C09108=1129.768,245.322,-69.072,-178.598,9.848,149.571
C09109=1129.764,245.570,-69.100,-178.596,9.851,149.571
C09110=1129.759,245.818,-69.127,-178.595,9.853,149.572
C09111=1129.756,246.067,-69.155,-178.594,9.855,149.572
C09112=1129.751,246.315,-69.183,-178.593,9.857,149.572
C09113=1129.747,246.564,-69.212,-178.591,9.859,149.572
C09114=1129.742,246.812,-69.239,-178.590,9.861,149.572
C09115=1129.738,247.060,-69.266,-178.588,9.864,149.572
C09116=1129.734,247.309,-69.295,-178.587,9.865,149.572
C09117=1129.729,247.557,-69.322,-178.583,9.870,149.572
C09118=1129.725,247.806,-69.350,-178.576,9.875,149.572
C09119=1129.721,248.054,-69.378,-178.568,9.881,149.571
C09120=1129.716,248.302,-69.406,-178.562,9.886,149.571
C09121=1129.711,248.551,-69.434,-178.555,9.891,149.570
C09122=1129.707,248.799,-69.462,-178.549,9.896,149.570
C09123=1129.703,249.048,-69.490,-178.543,9.900,149.569
C09124=1129.698,249.296,-69.518,-178.537,9.905,149.568
C09125=1129.694,249.545,-69.546,-178.532,9.909,149.568
C09126=1129.690,249.792,-69.574,-178.526,9.913,149.568
C09127=1129.686,250.041,-69.603,-178.521,9.917,149.567
C09128=1129.682,250.290,-69.631,-178.516,9.921,149.567
C09129=1129.678,250.538,-69.659,-178.512,9.925,149.567
C09130=1129.673,250.787,-69.688,-178.507,9.928,149.566
C09131=1129.669,251.034,-69.715,-178.503,9.931,149.566
C09132=1129.664,251.283,-69.744,-178.499,9.934,149.565
C09133=1129.660,251.531,-69.772,-178.495,9.937,149.565
C09134=1129.656,251.780,-69.801,-178.492,9.940,149.565
C09135=1129.652,252.028,-69.829,-178.488,9.943,149.565
C09136=1129.648,252.276,-69.857,-178.486,9.945,149.565
C09137=1129.643,252.525,-69.886,-178.483,9.947,149.565
C09138=1129.639,252.739,-69.910,-178.481,9.949,149.564
C09139=1129.635,252.953,-69.935,-178.479,9.951,149.564
C09140=1129.633,253.166,-69.960,-178.477,9.953,149.564
C09141=1129.628,253.379,-69.984,-178.476,9.955,149.564
C09142=1129.624,253.593,-70.008,-178.474,9.956,149.564
C09143=1129.620,253.807,-70.033,-178.474,9.957,149.564
C09144=1129.617,254.021,-70.058,-178.472,9.958,149.564
C09145=1129.613,254.235,-70.082,-178.472,9.959,149.564
C09146=1129.609,254.484,-70.110,-178.471,9.961,149.565
C09147=1129.605,254.732,-70.139,-178.471,9.962,149.565
C09148=1129.600,254.980,-70.167,-178.470,9.963,149.565
C09149=1129.596,255.229,-70.196,-178.471,9.963,149.565
C09150=1129.592,255.476,-70.224,-178.471,9.965,149.566
C09151=1129.587,255.725,-70.253,-178.472,9.966,149.566
C09152=1129.583,255.974,-70.281,-178.472,9.966,149.566
C09153=1129.579,256.221,-70.310,-178.469,9.969,149.566
C09154=1129.575,256.470,-70.338,-178.467,9.972,149.566
C09155=1129.570,256.719,-70.367,-178.464,9.975,149.566
C09156=1129.566,256.967,-70.395,-178.461,9.977,149.566
C09157=1129.562,257.215,-70.424,-178.458,9.980,149.566
C09158=1129.557,257.464,-70.453,-178.455,9.983,149.566
C09159=1129.553,257.712,-70.481,-178.451,9.986,149.566
C09160=1129.549,257.960,-70.510,-178.448,9.989,149.565
C09161=1129.545,258.209,-70.538,-178.446,9.992,149.565
C09162=1129.540,258.457,-70.567,-178.443,9.995,149.565
C09163=1129.536,258.705,-70.596,-178.439,9.998,149.565
C09164=1129.532,258.954,-70.624,-178.436,10.001,149.565
C09165=1129.527,259.201,-70.653,-178.433,10.004,149.565
C09166=1129.523,259.450,-70.682,-178.430,10.007,149.565
C09167=1129.519,259.698,-70.711,-178.427,10.010,149.565
C09168=1129.514,259.946,-70.739,-178.423,10.013,149.564
C09169=1129.510,260.195,-70.769,-178.420,10.016,149.564
C09170=1129.506,260.443,-70.797,-178.416,10.019,149.564
C09171=1129.502,260.691,-70.826,-178.413,10.022,149.564
C09172=1129.497,260.940,-70.855,-178.409,10.025,149.564
C09173=1129.493,261.188,-70.884,-178.406,10.028,149.564
C09174=1129.489,261.436,-70.912,-178.402,10.031,149.563
C09175=1129.485,261.685,-70.942,-178.399,10.034,149.563
C09176=1129.480,261.933,-70.970,-178.395,10.037,149.563
C09177=1129.476,262.181,-71.000,-178.392,10.041,149.563
C09178=1129.472,262.429,-71.028,-178.388,10.044,149.563
C09179=1129.468,262.678,-71.057,-178.385,10.047,149.563
C09180=1129.463,262.926,-71.086,-178.381,10.050,149.562
C09181=1129.459,263.174,-71.115,-178.377,10.053,149.562
C09182=1129.454,263.423,-71.144,-178.373,10.056,149.562
C09183=1129.451,263.671,-71.173,-178.369,10.060,149.562
C09184=1129.447,263.919,-71.203,-178.366,10.062,149.561
C09185=1129.442,264.168,-71.232,-178.362,10.065,149.561
C09186=1129.437,264.415,-71.261,-178.358,10.069,149.561
C09187=1129.433,264.664,-71.290,-178.355,10.071,149.561
C09188=1129.429,264.912,-71.320,-178.353,10.073,149.561
C09189=1129.425,265.161,-71.348,-178.350,10.076,149.560
C09190=1129.420,265.409,-71.378,-178.347,10.078,149.560
C09191=1129.416,265.657,-71.407,-178.346,10.080,149.560
C09192=1129.411,265.905,-71.436,-178.343,10.083,149.560
C09193=1129.408,266.153,-71.465,-178.340,10.085,149.560
C09194=1129.404,266.367,-71.491,-178.338,10.087,149.560
C09195=1129.400,266.581,-71.516,-178.336,10.089,149.560
C09196=1129.397,266.795,-71.541,-178.334,10.091,149.560
C09197=1129.393,267.008,-71.566,-178.331,10.093,149.560
C09198=1129.390,267.222,-71.591,-178.329,10.095,149.560
C09199=1129.385,267.435,-71.617,-178.327,10.097,149.560
C09200=1129.382,267.649,-71.642,-178.325,10.100,149.560
C09201=1129.378,267.863,-71.667,-178.323,10.102,149.560
C09202=1129.374,268.111,-71.696,-178.320,10.104,149.559
C09203=1129.370,268.359,-71.726,-178.317,10.106,149.559
C09204=1129.365,268.608,-71.755,-178.314,10.109,149.559
C09205=1129.361,268.856,-71.785,-178.312,10.112,149.559
C09206=1129.357,269.104,-71.814,-178.309,10.114,149.559
C09207=1129.353,269.352,-71.843,-178.306,10.117,149.559
C09208=1129.349,269.601,-71.873,-178.303,10.119,149.559
C09209=1129.345,269.849,-71.902,-178.301,10.121,149.559
C09210=1129.340,270.097,-71.932,-178.298,10.124,149.559
C09211=1129.336,270.346,-71.961,-178.295,10.127,149.558
C09212=1129.332,270.594,-71.991,-178.292,10.130,149.558
C09213=1129.328,270.841,-72.021,-178.290,10.132,149.558
C09214=1129.324,271.090,-72.050,-178.287,10.134,149.558
C09215=1129.319,271.338,-72.080,-178.284,10.137,149.558
C09216=1129.315,271.587,-72.110,-178.281,10.140,149.558
C09217=1129.311,271.835,-72.139,-178.278,10.143,149.558
C09218=1129.307,272.083,-72.169,-178.275,10.145,149.558
C09219=1129.302,272.331,-72.198,-178.272,10.148,149.558
C09220=1129.298,272.579,-72.228,-178.270,10.150,149.558
C09221=1129.294,272.827,-72.258,-178.267,10.153,149.557
C09222=1129.290,273.076,-72.287,-178.264,10.156,149.557
C09223=1129.285,273.324,-72.317,-178.261,10.158,149.557
C09224=1129.281,273.572,-72.347,-178.258,10.161,149.557
C09225=1129.277,273.820,-72.377,-178.255,10.164,149.557
C09226=1129.273,274.068,-72.406,-178.252,10.166,149.557
C09227=1129.269,274.317,-72.436,-178.249,10.169,149.557
C09228=1129.264,274.565,-72.466,-178.246,10.172,149.557
C09229=1129.260,274.813,-72.496,-178.243,10.174,149.556
C09230=1129.256,275.061,-72.525,-178.240,10.177,149.556
C09231=1129.252,275.309,-72.555,-178.236,10.181,149.556
C09232=1129.248,275.557,-72.585,-178.233,10.183,149.556
C09233=1129.243,275.806,-72.615,-178.230,10.186,149.556
C09234=1129.239,276.054,-72.645,-178.227,10.188,149.556
C09235=1129.235,276.301,-72.675,-178.224,10.191,149.555
C09236=1129.231,276.550,-72.704,-178.221,10.194,149.555
C09237=1129.226,276.798,-72.735,-178.217,10.197,149.555
C09238=1129.222,277.047,-72.765,-178.214,10.200,149.555
C09239=1129.218,277.294,-72.795,-178.211,10.202,149.555
C09240=1129.214,277.543,-72.825,-178.207,10.205,149.554
C09241=1129.210,277.791,-72.855,-178.205,10.208,149.554
C09242=1129.206,278.039,-72.885,-178.201,10.211,149.554
C09243=1129.201,278.287,-72.915,-178.198,10.213,149.554
C09244=1129.197,278.535,-72.945,-178.194,10.216,149.554
C09245=1129.193,278.783,-72.975,-178.191,10.219,149.554
C09246=1129.189,279.032,-73.005,-178.187,10.222,149.553
C09247=1129.185,279.280,-73.036,-178.184,10.225,149.553
C09248=1129.180,279.528,-73.065,-178.180,10.228,149.553
C09249=1129.176,279.776,-73.096,-178.177,10.230,149.553
C09250=1129.172,279.989,-73.121,-178.174,10.233,149.553
C09251=1129.169,280.203,-73.148,-178.171,10.236,149.552
C09252=1129.165,280.417,-73.174,-178.169,10.237,149.552
C09253=1129.162,280.630,-73.200,-178.166,10.240,149.552
C09254=1129.158,280.844,-73.226,-178.162,10.243,149.552
C09255=1129.154,281.057,-73.252,-178.159,10.245,149.552
C09256=1129.151,281.271,-73.278,-178.156,10.248,149.551
C09257=1129.147,281.484,-73.304,-178.153,10.250,149.551
C09258=1129.143,281.732,-73.334,-178.150,10.253,149.551
C09259=1129.139,281.981,-73.366,-178.147,10.255,149.551
C09260=1129.135,282.229,-73.395,-178.144,10.257,149.551
C09261=1129.130,282.477,-73.426,-178.141,10.260,149.551
C09262=1129.126,282.725,-73.456,-178.138,10.262,149.550
C09263=1129.122,282.973,-73.487,-178.135,10.265,149.550
C09264=1129.118,283.221,-73.516,-178.132,10.268,149.550
C09265=1129.113,283.469,-73.547,-178.129,10.270,149.550
C09266=1129.109,283.717,-73.577,-178.126,10.273,149.550
C09267=1129.105,283.965,-73.608,-178.122,10.276,149.549
C09268=1129.101,284.214,-73.639,-178.119,10.278,149.549
C09269=1129.097,284.461,-73.669,-178.117,10.280,149.549
C09270=1129.092,284.709,-73.700,-178.114,10.283,149.549
C09271=1129.088,284.958,-73.730,-178.111,10.286,149.549
C09272=1129.084,285.206,-73.761,-178.107,10.288,149.549
C09273=1129.080,285.454,-73.792,-178.104,10.291,149.548
C09274=1129.076,285.702,-73.822,-178.101,10.293,149.548
C09275=1129.072,285.951,-73.853,-178.098,10.296,149.548
C09276=1129.067,286.198,-73.884,-178.095,10.298,149.548
C09277=1129.063,286.446,-73.914,-178.092,10.301,149.548
C09278=1129.059,286.695,-73.945,-178.089,10.303,149.547
C09279=1129.055,286.943,-73.976,-178.086,10.306,149.547
C09280=1129.051,287.190,-74.006,-178.083,10.308,149.547
C09281=1129.047,287.439,-74.037,-178.080,10.311,149.547
C09282=1129.042,287.687,-74.068,-178.077,10.313,149.547
C09283=1129.038,287.935,-74.098,-178.074,10.316,149.547
C09284=1129.034,288.183,-74.129,-178.071,10.319,149.546
C09285=1129.030,288.431,-74.161,-178.067,10.321,149.546
C09286=1129.026,288.678,-74.191,-178.064,10.324,149.546
C09287=1129.022,288.927,-74.222,-178.061,10.326,149.546
C09288=1129.017,289.175,-74.253,-178.058,10.329,149.546
C09289=1129.013,289.423,-74.283,-178.055,10.332,149.546
C09290=1129.009,289.671,-74.314,-178.052,10.334,149.545
C09291=1129.005,289.919,-74.345,-178.050,10.336,149.545
C09292=1129.001,290.167,-74.377,-178.046,10.339,149.545
C09293=1128.996,290.415,-74.407,-178.043,10.341,149.545
C09294=1128.992,290.663,-74.438,-178.040,10.344,149.545
C09295=1128.989,290.911,-74.469,-178.037,10.346,149.545
C09296=1128.984,291.159,-74.500,-178.034,10.349,149.544
C09297=1128.980,291.407,-74.531,-178.031,10.352,149.544
C09298=1128.976,291.655,-74.562,-178.027,10.354,149.544
C09299=1128.972,291.904,-74.593,-178.025,10.357,149.544
C09300=1128.967,292.151,-74.625,-178.021,10.359,149.544
C09301=1128.964,292.400,-74.655,-178.018,10.362,149.543
C09302=1128.959,292.648,-74.686,-178.016,10.364,149.543
C09303=1128.955,292.895,-74.717,-178.013,10.366,149.543
C09304=1128.951,293.144,-74.748,-178.010,10.369,149.543
C09305=1128.947,293.391,-74.780,-178.006,10.372,149.543
C09306=1128.943,293.605,-74.807,-178.003,10.374,149.543
C09307=1128.940,293.819,-74.834,-178.001,10.376,149.542
C09308=1128.936,294.032,-74.860,-177.998,10.378,149.542
C09309=1128.933,294.246,-74.887,-177.995,10.381,149.542
C09310=1128.929,294.458,-74.914,-177.993,10.383,149.542
C09311=1128.926,294.672,-74.941,-177.990,10.384,149.542
C09312=1128.922,294.886,-74.968,-177.988,10.387,149.542
C09313=1128.918,295.099,-74.994,-177.985,10.389,149.541
C09314=1128.914,295.347,-75.026,-177.982,10.392,149.541
C09315=1128.910,295.595,-75.057,-177.979,10.394,149.541
C09316=1128.906,295.843,-75.089,-177.976,10.397,149.541
C09317=1128.902,296.091,-75.120,-177.973,10.400,149.541
C09318=1128.898,296.339,-75.152,-177.969,10.402,149.540
C09319=1128.893,296.587,-75.182,-177.966,10.405,149.540
C09320=1128.890,296.835,-75.214,-177.963,10.407,149.540
C09321=1128.886,297.083,-75.246,-177.960,10.410,149.540
C09322=1128.881,297.331,-75.277,-177.957,10.412,149.540
C09323=1128.877,297.579,-75.309,-177.954,10.414,149.540
C09324=1128.873,297.827,-75.339,-177.951,10.417,149.539
C09325=1128.869,298.075,-75.371,-177.948,10.420,149.539
C09326=1128.865,298.322,-75.403,-177.945,10.422,149.539
C09327=1128.861,298.571,-75.434,-177.942,10.425,149.539
C09328=1128.857,298.818,-75.465,-177.939,10.427,149.539
C09329=1128.853,299.066,-75.497,-177.936,10.430,149.539
C09330=1128.849,299.314,-75.529,-177.932,10.432,149.538
C09331=1128.844,299.563,-75.560,-177.929,10.435,149.538
C09332=1128.840,299.811,-75.592,-177.926,10.438,149.538
C09333=1128.836,300.058,-75.624,-177.923,10.440,149.538
C09334=1128.832,300.306,-75.655,-177.920,10.443,149.538
C09335=1128.828,300.555,-75.687,-177.918,10.445,149.538
C09336=1128.824,300.802,-75.718,-177.914,10.447,149.537
C09337=1128.819,301.050,-75.751,-177.911,10.450,149.537
C09338=1128.816,301.298,-75.782,-177.908,10.452,149.537
C09339=1128.811,301.546,-75.814,-177.905,10.455,149.537
C09340=1128.807,301.794,-75.845,-177.902,10.458,149.537
C09341=1128.803,302.042,-75.876,-177.899,10.460,149.536
C09342=1128.799,302.290,-75.909,-177.895,10.463,149.536
C09343=1128.795,302.538,-75.941,-177.892,10.466,149.536
C09344=1128.790,302.785,-75.972,-177.889,10.468,149.536
C09345=1128.787,303.033,-76.004,-177.886,10.471,149.536
C09346=1128.782,303.282,-76.037,-177.883,10.473,149.536
C09347=1128.778,303.529,-76.068,-177.880,10.476,149.535
C09348=1128.774,303.777,-76.100,-177.877,10.478,149.535
C09349=1128.771,304.025,-76.132,-177.874,10.480,149.535
C09350=1128.766,304.274,-76.164,-177.871,10.483,149.535
C09351=1128.762,304.521,-76.196,-177.868,10.485,149.535
C09352=1128.758,304.769,-76.227,-177.865,10.488,149.534
C09353=1128.754,305.017,-76.260,-177.861,10.490,149.534
C09354=1128.749,305.265,-76.291,-177.858,10.493,149.534
C09355=1128.746,305.513,-76.323,-177.855,10.496,149.534
C09356=1128.741,305.761,-76.356,-177.852,10.498,149.534
C09357=1128.738,306.009,-76.388,-177.849,10.501,149.534
C09358=1128.733,306.256,-76.419,-177.846,10.504,149.533
C09359=1128.729,306.505,-76.451,-177.843,10.506,149.533
C09360=1128.725,306.753,-76.483,-177.839,10.508,149.533
C09361=1128.721,307.001,-76.516,-177.836,10.511,149.533
C09362=1128.717,307.214,-76.543,-177.834,10.513,149.533
C09363=1128.714,307.427,-76.571,-177.831,10.515,149.532
C09364=1128.710,307.640,-76.599,-177.828,10.518,149.532
C09365=1128.707,307.854,-76.626,-177.826,10.519,149.532
C09366=1128.703,308.067,-76.654,-177.823,10.522,149.532
C09367=1128.699,308.280,-76.682,-177.820,10.524,149.532
C09368=1128.696,308.493,-76.709,-177.818,10.526,149.532
C09369=1128.693,308.706,-76.737,-177.815,10.529,149.532
C09370=1128.689,308.954,-76.769,-177.812,10.531,149.531
C09371=1128.684,309.203,-76.802,-177.809,10.534,149.531
C09372=1128.681,309.450,-76.834,-177.806,10.535,149.531
C09373=1128.676,309.698,-76.866,-177.803,10.538,149.531
C09374=1128.672,309.946,-76.898,-177.800,10.541,149.531
C09375=1128.668,310.193,-76.931,-177.797,10.543,149.530
C09376=1128.664,310.442,-76.963,-177.793,10.546,149.530
C09377=1128.660,310.690,-76.996,-177.790,10.549,149.530
C09378=1128.657,310.937,-77.028,-177.787,10.551,149.530
C09379=1128.651,311.185,-77.060,-177.784,10.553,149.530
C09380=1128.648,311.433,-77.092,-177.781,10.556,149.530
C09381=1128.644,311.681,-77.125,-177.777,10.559,149.529
C09382=1128.640,311.929,-77.157,-177.775,10.561,149.529
C09383=1128.636,312.176,-77.190,-177.771,10.564,149.529
C09384=1128.631,312.425,-77.223,-177.768,10.566,149.529
C09385=1128.628,312.672,-77.255,-177.765,10.569,149.529
C09386=1128.624,312.921,-77.288,-177.762,10.571,149.528
C09387=1128.620,313.167,-77.320,-177.759,10.574,149.528
C09388=1128.615,313.416,-77.352,-177.756,10.576,149.528
C09389=1128.611,313.663,-77.385,-177.753,10.578,149.528
C09390=1128.607,313.911,-77.417,-177.750,10.581,149.528
C09391=1128.603,314.159,-77.450,-177.746,10.584,149.527
C09392=1128.599,314.408,-77.483,-177.744,10.586,149.527
C09393=1128.595,314.655,-77.515,-177.740,10.589,149.527
C09394=1128.591,314.903,-77.549,-177.737,10.591,149.527
C09395=1128.587,315.151,-77.581,-177.734,10.594,149.527
C09396=1128.583,315.398,-77.614,-177.731,10.596,149.527
C09397=1128.579,315.647,-77.646,-177.728,10.599,149.526
C09398=1128.575,315.895,-77.679,-177.724,10.602,149.526
C09399=1128.571,316.142,-77.712,-177.721,10.604,149.526
C09400=1128.567,316.390,-77.744,-177.718,10.607,149.526
C09401=1128.563,316.638,-77.777,-177.715,10.609,149.526
C09402=1128.559,316.885,-77.810,-177.711,10.612,149.525
C09403=1128.555,317.133,-77.843,-177.708,10.615,149.525
C09404=1128.551,317.382,-77.876,-177.706,10.616,149.525
C09405=1128.547,317.629,-77.909,-177.703,10.619,149.525
C09406=1128.543,317.877,-77.941,-177.700,10.621,149.525
C09407=1128.539,318.124,-77.974,-177.696,10.624,149.524
C09408=1128.535,318.372,-78.008,-177.693,10.627,149.524
C09409=1128.530,318.620,-78.040,-177.690,10.629,149.524
C09410=1128.526,318.868,-78.073,-177.687,10.631,149.524
C09411=1128.523,319.116,-78.106,-177.684,10.634,149.524
C09412=1128.519,319.363,-78.139,-177.680,10.637,149.524
C09413=1128.515,319.611,-78.172,-177.677,10.639,149.523
C09414=1128.510,319.859,-78.205,-177.674,10.642,149.523
C09415=1128.506,320.107,-78.238,-177.671,10.644,149.523
C09416=1128.502,320.355,-78.271,-177.668,10.647,149.523
C09417=1128.499,320.602,-78.303,-177.665,10.650,149.523
C09418=1128.495,320.815,-78.332,-177.662,10.652,149.523
C09419=1128.491,321.028,-78.361,-177.659,10.654,149.522
C09420=1128.488,321.242,-78.389,-177.657,10.656,149.522
C09421=1128.485,321.454,-78.418,-177.654,10.658,149.522
C09422=1128.481,321.668,-78.446,-177.651,10.660,149.522
C09423=1128.478,321.881,-78.475,-177.648,10.662,149.522
C09424=1128.474,322.093,-78.503,-177.645,10.665,149.522
C09425=1128.470,322.307,-78.532,-177.643,10.667,149.521
C09426=1128.467,322.555,-78.565,-177.640,10.669,149.521
C09427=1128.463,322.803,-78.598,-177.636,10.672,149.521
C09428=1128.459,323.050,-78.631,-177.634,10.675,149.521
C09429=1128.455,323.298,-78.664,-177.630,10.677,149.521
C09430=1128.451,323.545,-78.698,-177.627,10.679,149.520
C09431=1128.447,323.793,-78.731,-177.624,10.682,149.520
C09432=1128.443,324.041,-78.764,-177.621,10.685,149.520
C09433=1128.439,324.289,-78.798,-177.618,10.686,149.520
C09434=1128.435,324.537,-78.831,-177.615,10.689,149.520
C09435=1128.431,324.785,-78.864,-177.612,10.692,149.519
C09436=1128.427,325.032,-78.897,-177.608,10.694,149.519
C09437=1128.423,325.280,-78.931,-177.605,10.696,149.519
C09438=1128.419,325.527,-78.964,-177.602,10.699,149.519
C09439=1128.415,325.775,-78.997,-177.599,10.702,149.519
C09440=1128.411,326.024,-79.032,-177.595,10.704,149.518
C09441=1128.407,326.271,-79.065,-177.593,10.707,149.518
C09442=1128.403,326.519,-79.099,-177.589,10.709,149.518
C09443=1128.398,326.766,-79.132,-177.586,10.712,149.518
C09444=1128.394,327.014,-79.165,-177.583,10.715,149.518
C09445=1128.391,327.262,-79.199,-177.580,10.717,149.518
C09446=1128.387,327.510,-79.232,-177.576,10.719,149.517
C09447=1128.383,327.757,-79.265,-177.573,10.722,149.517
C09448=1128.379,328.004,-79.299,-177.570,10.725,149.517
C09449=1128.374,328.252,-79.333,-177.567,10.727,149.517
C09450=1128.371,328.500,-79.367,-177.563,10.730,149.517
C09451=1128.367,328.748,-79.400,-177.561,10.732,149.516
C09452=1128.363,328.996,-79.434,-177.557,10.735,149.516
C09453=1128.359,329.243,-79.467,-177.555,10.736,149.516
C09454=1128.355,329.491,-79.501,-177.552,10.739,149.516
C09455=1128.351,329.739,-79.535,-177.548,10.742,149.516
C09456=1128.346,329.986,-79.569,-177.545,10.744,149.515
C09457=1128.343,330.233,-79.602,-177.542,10.747,149.515
C09458=1128.339,330.482,-79.636,-177.539,10.749,149.515
C09459=1128.335,330.729,-79.670,-177.535,10.752,149.515
C09460=1128.330,330.977,-79.704,-177.532,10.754,149.515
C09461=1128.327,331.225,-79.738,-177.529,10.757,149.515
C09462=1128.323,331.473,-79.771,-177.526,10.759,149.514
C09463=1128.319,331.720,-79.805,-177.523,10.762,149.514
C09464=1128.314,331.968,-79.839,-177.519,10.764,149.514
C09465=1128.311,332.216,-79.873,-177.516,10.767,149.514
C09466=1128.307,332.463,-79.907,-177.513,10.770,149.514
C09467=1128.302,332.711,-79.940,-177.510,10.772,149.513
C09468=1128.299,332.959,-79.975,-177.506,10.774,149.513
C09469=1128.295,333.206,-80.009,-177.503,10.777,149.513
C09470=1128.290,333.454,-80.042,-177.500,10.780,149.513
C09471=1128.287,333.701,-80.077,-177.497,10.782,149.512
C09472=1128.283,333.949,-80.110,-177.493,10.785,149.512
C09473=1128.279,334.197,-80.145,-177.491,10.787,149.512
C09474=1128.276,334.410,-80.174,-177.488,10.789,149.512
C09475=1128.272,334.622,-80.203,-177.486,10.791,149.512
C09476=1128.269,334.835,-80.232,-177.482,10.794,149.512
C09477=1128.266,335.048,-80.262,-177.480,10.796,149.512
C09478=1128.262,335.262,-80.291,-177.477,10.798,149.511
C09479=1128.258,335.474,-80.320,-177.474,10.800,149.511
C09480=1128.255,335.687,-80.349,-177.472,10.802,149.511
C09481=1128.252,335.900,-80.379,-177.468,10.804,149.511
C09482=1128.248,336.148,-80.414,-177.465,10.807,149.511
C09483=1128.244,336.396,-80.447,-177.462,10.809,149.510
C09484=1128.240,336.643,-80.481,-177.459,10.812,149.510
C09485=1128.236,336.891,-80.515,-177.455,10.814,149.510
C09486=1128.233,337.138,-80.550,-177.453,10.817,149.510
C09487=1128.228,337.386,-80.584,-177.450,10.819,149.510
C09488=1128.225,337.634,-80.618,-177.446,10.821,149.509
C09489=1128.220,337.881,-80.653,-177.443,10.824,149.509
C09490=1128.217,338.129,-80.687,-177.440,10.826,149.509
C09491=1128.212,338.376,-80.722,-177.437,10.829,149.509
C09492=1128.209,338.623,-80.755,-177.434,10.831,149.509
C09493=1128.205,338.872,-80.790,-177.430,10.834,149.508
C09494=1128.201,339.119,-80.824,-177.427,10.836,149.508
C09495=1128.197,339.367,-80.859,-177.424,10.839,149.508
C09496=1128.192,339.614,-80.893,-177.421,10.841,149.508
C09497=1128.189,339.862,-80.928,-177.417,10.844,149.508
C09498=1128.184,340.109,-80.962,-177.414,10.846,149.507
C09499=1128.181,340.357,-80.996,-177.411,10.849,149.507
C09500=1128.177,340.605,-81.031,-177.408,10.852,149.507
C09501=1128.173,340.853,-81.066,-177.405,10.854,149.507
C09502=1128.169,341.100,-81.100,-177.401,10.857,149.507
C09503=1128.165,341.348,-81.134,-177.398,10.859,149.506
C09504=1128.161,341.595,-81.168,-177.395,10.861,149.506
C09505=1128.157,341.843,-81.204,-177.391,10.864,149.506
C09506=1128.153,342.090,-81.238,-177.388,10.867,149.506
C09507=1128.150,342.338,-81.272,-177.385,10.869,149.506
C09508=1128.145,342.585,-81.307,-177.382,10.872,149.505
C09509=1128.141,342.833,-81.342,-177.378,10.874,149.505
C09510=1128.137,343.080,-81.376,-177.375,10.876,149.505
C09511=1128.134,343.328,-81.411,-177.372,10.878,149.505
C09512=1128.129,343.575,-81.446,-177.370,10.881,149.505
C09513=1128.125,343.824,-81.481,-177.366,10.883,149.504
C09514=1128.121,344.070,-81.515,-177.363,10.886,149.504
C09515=1128.117,344.318,-81.550,-177.360,10.888,149.504
C09516=1128.114,344.566,-81.585,-177.356,10.891,149.504
C09517=1128.110,344.813,-81.619,-177.353,10.893,149.503
C09518=1128.106,345.061,-81.654,-177.350,10.896,149.503
C09519=1128.101,345.308,-81.689,-177.347,10.898,149.503
C09520=1128.098,345.556,-81.724,-177.343,10.901,149.503
C09521=1128.094,345.804,-81.759,-177.340,10.903,149.503
C09522=1128.090,346.050,-81.794,-177.337,10.906,149.502
C09523=1128.086,346.299,-81.828,-177.333,10.908,149.502
C09524=1128.082,346.546,-81.863,-177.330,10.911,149.502
C09525=1128.078,346.793,-81.898,-177.327,10.914,149.502
C09526=1128.074,347.042,-81.933,-177.324,10.916,149.502
C09527=1128.071,347.288,-81.968,-177.321,10.918,149.501
C09528=1128.067,347.536,-82.003,-177.317,10.921,149.501
C09529=1128.063,347.784,-82.038,-177.314,10.923,149.501
C09530=1128.059,347.996,-82.068,-177.312,10.925,149.501
C09531=1128.056,348.209,-82.098,-177.308,10.928,149.501
C09532=1128.052,348.422,-82.129,-177.306,10.930,149.500
C09533=1128.050,348.635,-82.159,-177.303,10.932,149.500
C09534=1128.046,348.847,-82.189,-177.300,10.934,149.500
C09535=1128.043,349.061,-82.219,-177.297,10.936,149.500
C09536=1128.039,349.273,-82.249,-177.295,10.938,149.500
C09537=1128.036,349.486,-82.279,-177.292,10.940,149.500
C09538=1128.031,349.734,-82.314,-177.289,10.943,149.499
C09539=1128.028,349.981,-82.350,-177.285,10.946,149.499
C09540=1128.024,350.229,-82.385,-177.281,10.948,149.499
C09541=1128.020,350.477,-82.420,-177.278,10.950,149.499
C09542=1128.016,350.723,-82.455,-177.274,10.954,149.498
C09543=1128.012,350.971,-82.491,-177.270,10.956,149.498
C09544=1128.008,351.219,-82.525,-177.266,10.959,149.498
C09545=1128.004,351.466,-82.561,-177.263,10.962,149.498
C09546=1128.000,351.713,-82.596,-177.259,10.964,149.497
C09547=1127.997,351.961,-82.632,-177.256,10.966,149.497
C09548=1127.993,352.208,-82.667,-177.252,10.970,149.497
C09549=1127.988,352.456,-82.702,-177.248,10.972,149.496
C09550=1127.985,352.703,-82.737,-177.245,10.974,149.496
C09551=1127.981,352.951,-82.773,-177.241,10.978,149.496
C09552=1127.977,353.198,-82.808,-177.238,10.980,149.496
C09553=1127.974,353.446,-82.844,-177.234,10.982,149.495
C09554=1127.969,353.693,-82.879,-177.231,10.985,149.495
C09555=1127.966,353.941,-82.914,-177.227,10.988,149.495
C09556=1127.962,354.188,-82.949,-177.224,10.990,149.495
C09557=1127.958,354.436,-82.985,-177.220,10.992,149.494
C09558=1127.955,354.683,-83.021,-177.217,10.995,149.494
C09559=1127.950,354.930,-83.056,-177.213,10.998,149.494
C09560=1127.947,355.178,-83.091,-177.209,11.001,149.494
C09561=1127.943,355.425,-83.127,-177.206,11.003,149.493
C09562=1127.939,355.673,-83.163,-177.202,11.005,149.493
C09563=1127.935,355.920,-83.199,-177.199,11.008,149.493
C09564=1127.931,356.168,-83.234,-177.196,11.010,149.493
C09565=1127.927,356.415,-83.269,-177.191,11.013,149.492
C09566=1127.923,356.662,-83.305,-177.188,11.015,149.492
C09567=1127.920,356.909,-83.341,-177.185,11.018,149.492
C09568=1127.916,357.157,-83.377,-177.181,11.020,149.492
C09569=1127.912,357.404,-83.413,-177.178,11.023,149.491
C09570=1127.908,357.652,-83.448,-177.174,11.025,149.491
C09571=1127.905,357.899,-83.484,-177.171,11.027,149.491
C09572=1127.901,358.147,-83.519,-177.167,11.030,149.490
C09573=1127.896,358.395,-83.556,-177.163,11.033,149.490
C09574=1127.893,358.641,-83.591,-177.160,11.035,149.490
C09575=1127.889,358.888,-83.627,-177.157,11.038,149.490
C09576=1127.885,359.136,-83.663,-177.153,11.040,149.489
C09577=1127.881,359.384,-83.699,-177.150,11.042,149.489
C09578=1127.877,359.631,-83.734,-177.147,11.045,149.489
C09579=1127.874,359.878,-83.771,-177.143,11.047,149.489
C09580=1127.869,360.126,-83.807,-177.140,11.049,149.488
C09581=1127.866,360.373,-83.842,-177.136,11.052,149.488
C09582=1127.862,360.620,-83.878,-177.133,11.054,149.488
C09583=1127.859,360.868,-83.914,-177.130,11.057,149.488
C09584=1127.854,361.116,-83.950,-177.126,11.059,149.487
C09585=1127.851,361.362,-83.986,-177.123,11.061,149.487
C09586=1127.848,361.576,-84.017,-177.120,11.063,149.487
C09587=1127.844,361.788,-84.048,-177.117,11.066,149.487
C09588=1127.841,362.000,-84.079,-177.114,11.068,149.486
C09589=1127.838,362.213,-84.110,-177.111,11.070,149.486
C09590=1127.834,362.426,-84.141,-177.108,11.072,149.486
C09591=1127.831,362.639,-84.172,-177.105,11.074,149.486
C09592=1127.828,362.851,-84.203,-177.102,11.076,149.486
C09593=1127.825,363.063,-84.234,-177.100,11.078,149.485
C09594=1127.820,363.311,-84.271,-177.096,11.080,149.485
C09595=1127.817,363.558,-84.307,-177.093,11.083,149.485
C09596=1127.813,363.806,-84.342,-177.090,11.085,149.485
C09597=1127.809,364.053,-84.379,-177.086,11.087,149.484
C09598=1127.806,364.300,-84.415,-177.083,11.090,149.484
C09599=1127.801,364.548,-84.452,-177.079,11.092,149.484
C09600=1127.798,364.795,-84.487,-177.076,11.095,149.484
C09601=1127.794,365.042,-84.524,-177.073,11.097,149.483
C09602=1127.791,365.290,-84.561,-177.070,11.100,149.483
C09603=1127.787,365.538,-84.597,-177.066,11.102,149.483
C09604=1127.783,365.784,-84.633,-177.063,11.103,149.483
C09605=1127.779,366.032,-84.669,-177.060,11.106,149.482
C09606=1127.775,366.279,-84.706,-177.057,11.108,149.482
C09607=1127.771,366.526,-84.742,-177.053,11.111,149.482
C09608=1127.768,366.774,-84.778,-177.050,11.113,149.482
C09609=1127.764,367.021,-84.815,-177.047,11.116,149.481
C09610=1127.760,367.268,-84.851,-177.043,11.118,149.481
C09611=1127.756,367.515,-84.888,-177.041,11.120,149.481
C09612=1127.752,367.763,-84.924,-177.037,11.122,149.481
C09613=1127.748,368.010,-84.960,-177.034,11.125,149.480
C09614=1127.745,368.258,-84.998,-177.030,11.127,149.480
C09615=1127.742,368.505,-85.034,-177.027,11.130,149.480
C09616=1127.737,368.752,-85.070,-177.024,11.132,149.480
C09617=1127.733,369.000,-85.107,-177.021,11.134,149.480
C09618=1127.730,369.246,-85.143,-177.018,11.136,149.479
C09619=1127.726,369.494,-85.180,-177.015,11.139,149.479
C09620=1127.721,369.741,-85.217,-177.011,11.141,149.479
C09621=1127.719,369.988,-85.253,-177.008,11.144,149.479
C09622=1127.714,370.236,-85.290,-177.005,11.145,149.478
C09623=1127.710,370.483,-85.326,-177.002,11.148,149.478
C09624=1127.707,370.730,-85.363,-176.999,11.150,149.478
C09625=1127.703,370.978,-85.400,-176.995,11.153,149.478
C09626=1127.699,371.225,-85.436,-176.993,11.154,149.478
C09627=1127.696,371.472,-85.473,-176.990,11.157,149.478
C09628=1127.692,371.719,-85.510,-176.986,11.160,149.477
C09629=1127.688,371.967,-85.547,-176.983,11.162,149.477
C09630=1127.684,372.214,-85.583,-176.981,11.164,149.477
C09631=1127.680,372.461,-85.620,-176.977,11.166,149.477
C09632=1127.677,372.709,-85.657,-176.974,11.169,149.476
C09633=1127.673,372.956,-85.694,-176.971,11.171,149.476
C09634=1127.669,373.203,-85.730,-176.968,11.173,149.476
C09635=1127.665,373.450,-85.767,-176.965,11.176,149.476
C09636=1127.662,373.698,-85.804,-176.962,11.178,149.476
C09637=1127.658,373.945,-85.841,-176.958,11.181,149.476
C09638=1127.654,374.192,-85.878,-176.956,11.182,149.475
C09639=1127.651,374.438,-85.915,-176.952,11.185,149.475
C09640=1127.647,374.686,-85.952,-176.950,11.188,149.475
C09641=1127.643,374.934,-85.989,-176.947,11.189,149.475
C09642=1127.640,375.146,-86.020,-176.944,11.192,149.475
C09643=1127.636,375.358,-86.053,-176.941,11.194,149.475
C09644=1127.633,375.571,-86.084,-176.939,11.196,149.474
C09645=1127.630,375.784,-86.116,-176.936,11.198,149.474
C09646=1127.627,375.996,-86.148,-176.934,11.200,149.474
C09647=1127.624,376.209,-86.179,-176.931,11.201,149.474
C09648=1127.620,376.421,-86.212,-176.929,11.204,149.474
C09649=1127.617,376.634,-86.243,-176.926,11.206,149.474
C09650=1127.613,376.881,-86.280,-176.924,11.208,149.474
C09651=1127.609,377.128,-86.318,-176.920,11.210,149.474
C09652=1127.605,377.375,-86.355,-176.917,11.213,149.473
C09653=1127.602,377.623,-86.392,-176.915,11.215,149.473
C09654=1127.598,377.869,-86.429,-176.911,11.217,149.473
C09655=1127.594,378.116,-86.466,-176.909,11.220,149.473
C09656=1127.590,378.364,-86.503,-176.906,11.222,149.473
C09657=1127.587,378.611,-86.541,-176.903,11.225,149.473
C09658=1127.583,378.858,-86.578,-176.900,11.227,149.473
C09659=1127.579,379.106,-86.615,-176.897,11.229,149.473
C09660=1127.576,379.352,-86.652,-176.894,11.232,149.472
C09661=1127.572,379.599,-86.689,-176.892,11.234,149.472
C09662=1127.569,379.847,-86.727,-176.889,11.236,149.472
C09663=1127.565,380.094,-86.764,-176.886,11.239,149.472
C09664=1127.561,380.341,-86.801,-176.883,11.241,149.472
C09665=1127.557,380.588,-86.838,-176.880,11.244,149.472
C09666=1127.553,380.835,-86.875,-176.877,11.246,149.472
C09667=1127.550,381.083,-86.913,-176.875,11.248,149.472
C09668=1127.545,381.330,-86.951,-176.872,11.251,149.472
C09669=1127.541,381.577,-86.988,-176.869,11.253,149.471
C09670=1127.538,381.825,-87.026,-176.866,11.255,149.471
C09671=1127.534,382.071,-87.063,-176.863,11.258,149.471
C09672=1127.531,382.319,-87.100,-176.861,11.260,149.471
C09673=1127.527,382.566,-87.138,-176.858,11.263,149.471
C09674=1127.523,382.813,-87.175,-176.855,11.265,149.471
C09675=1127.520,383.060,-87.213,-176.852,11.268,149.471
C09676=1127.516,383.307,-87.250,-176.850,11.270,149.471
C09677=1127.512,383.555,-87.287,-176.848,11.272,149.471
C09678=1127.509,383.801,-87.325,-176.846,11.274,149.471
C09679=1127.504,384.048,-87.362,-176.845,11.276,149.471
C09680=1127.501,384.296,-87.400,-176.843,11.278,149.471
C09681=1127.497,384.543,-87.438,-176.842,11.280,149.471
C09682=1127.493,384.790,-87.475,-176.840,11.281,149.471
C09683=1127.489,385.037,-87.513,-176.839,11.283,149.472
C09684=1127.486,385.284,-87.551,-176.837,11.285,149.472
C09685=1127.482,385.532,-87.588,-176.836,11.287,149.472
C09686=1127.479,385.779,-87.626,-176.834,11.289,149.472
C09687=1127.475,386.025,-87.663,-176.833,11.291,149.472
C09688=1127.472,386.273,-87.700,-176.831,11.293,149.472
C09689=1127.467,386.520,-87.739,-176.830,11.294,149.472
C09690=1127.463,386.767,-87.776,-176.829,11.296,149.472
C09691=1127.460,387.014,-87.814,-176.827,11.299,149.473
C09692=1127.456,387.261,-87.851,-176.826,11.300,149.473
C09693=1127.453,387.508,-87.889,-176.824,11.303,149.473
C09694=1127.449,387.755,-87.926,-176.823,11.305,149.473
C09695=1127.445,388.003,-87.965,-176.822,11.307,149.473
C09696=1127.441,388.250,-88.002,-176.820,11.309,149.473
C09697=1127.438,388.497,-88.040,-176.819,11.311,149.474
C09698=1127.434,388.709,-88.072,-176.818,11.312,149.474
C09699=1127.432,388.921,-88.104,-176.817,11.315,149.474
C09700=1127.428,389.134,-88.137,-176.816,11.317,149.474
C09701=1127.425,389.346,-88.170,-176.815,11.318,149.474
C09702=1127.423,389.559,-88.202,-176.814,11.320,149.475
C09703=1127.419,389.771,-88.234,-176.813,11.322,149.475
C09704=1127.416,389.984,-88.267,-176.812,11.324,149.475
C09705=1127.413,390.196,-88.299,-176.811,11.326,149.475
C09706=1127.408,390.442,-88.337,-176.809,11.328,149.476
C09707=1127.405,390.690,-88.374,-176.808,11.330,149.476
C09708=1127.402,390.938,-88.412,-176.807,11.333,149.476
C09709=1127.398,391.184,-88.450,-176.806,11.335,149.477
C09710=1127.394,391.432,-88.488,-176.805,11.338,149.477
C09711=1127.390,391.678,-88.526,-176.804,11.339,149.477
C09712=1127.387,391.926,-88.564,-176.803,11.342,149.478
C09713=1127.383,392.172,-88.602,-176.802,11.344,149.478
C09714=1127.380,392.419,-88.639,-176.800,11.347,149.478
C09715=1127.375,392.667,-88.677,-176.800,11.349,149.479
C09716=1127.372,392.914,-88.715,-176.798,11.352,149.479
C09717=1127.368,393.161,-88.752,-176.798,11.354,149.480
C09718=1127.364,393.408,-88.791,-176.796,11.357,149.480
C09719=1127.361,393.655,-88.829,-176.795,11.360,149.480
C09720=1127.357,393.902,-88.867,-176.795,11.362,149.481
C09721=1127.354,394.149,-88.904,-176.793,11.365,149.481
C09722=1127.350,394.396,-88.943,-176.793,11.367,149.482
C09723=1127.346,394.644,-88.981,-176.791,11.370,149.482
C09724=1127.343,394.890,-89.018,-176.791,11.372,149.482
C09725=1127.339,395.138,-89.057,-176.790,11.375,149.483
C09726=1127.335,395.384,-89.094,-176.789,11.378,149.483
C09727=1127.332,395.632,-89.132,-176.788,11.380,149.484
C09728=1127.327,395.878,-89.170,-176.787,11.383,149.484
C09729=1127.324,396.126,-89.208,-176.786,11.386,149.485
C09730=1127.320,396.372,-89.246,-176.786,11.388,149.485
C09731=1127.316,396.620,-89.284,-176.785,11.391,149.486
C09732=1127.313,396.867,-89.322,-176.785,11.394,149.486
C09733=1127.309,397.114,-89.360,-176.784,11.397,149.487
C09734=1127.305,397.361,-89.398,-176.782,11.400,149.488
C09735=1127.302,397.608,-89.436,-176.782,11.403,149.488
C09736=1127.298,397.855,-89.475,-176.781,11.406,149.489
C09737=1127.295,398.103,-89.512,-176.781,11.409,149.489
C09738=1127.291,398.349,-89.550,-176.779,11.412,149.490
C09739=1127.287,398.597,-89.589,-176.779,11.415,149.491
C09740=1127.283,398.843,-89.626,-176.779,11.418,149.491
C09741=1127.280,399.091,-89.664,-176.778,11.421,149.492
C09742=1127.276,399.338,-89.703,-176.778,11.423,149.492
C09743=1127.272,399.584,-89.741,-176.777,11.427,149.493
C09744=1127.268,399.832,-89.779,-176.776,11.430,149.494
C09745=1127.265,400.078,-89.817,-176.775,11.433,149.494
C09746=1127.262,400.326,-89.855,-176.775,11.436,149.495
C09747=1127.258,400.573,-89.894,-176.775,11.439,149.496
C09748=1127.254,400.820,-89.931,-176.774,11.443,149.496
C09749=1127.250,401.067,-89.970,-176.774,11.446,149.497
C09750=1127.247,401.314,-90.008,-176.773,11.450,149.498
C09751=1127.243,401.561,-90.046,-176.773,11.452,149.499
C09752=1127.239,401.808,-90.084,-176.773,11.456,149.500
C09753=1127.236,402.055,-90.122,-176.772,11.459,149.500
C09754=1127.233,402.268,-90.155,-176.772,11.462,149.501
C09755=1127.229,402.480,-90.188,-176.771,11.465,149.502
C09756=1127.226,402.692,-90.221,-176.771,11.468,149.502
C09757=1127.222,402.904,-90.253,-176.770,11.471,149.503
C09758=1127.220,403.117,-90.287,-176.770,11.474,149.504
C09759=1127.216,403.329,-90.320,-176.770,11.477,149.504
C09760=1127.214,403.541,-90.352,-176.770,11.480,149.505
C09761=1127.211,403.753,-90.385,-176.769,11.483,149.506
C09762=1127.207,404.000,-90.423,-176.769,11.487,149.507
C09763=1127.203,404.248,-90.461,-176.769,11.490,149.507
C09764=1127.199,404.494,-90.500,-176.769,11.493,149.508
C09765=1127.196,404.741,-90.538,-176.769,11.497,149.509
C09766=1127.192,404.989,-90.577,-176.769,11.501,149.510
C09767=1127.188,405.235,-90.614,-176.768,11.505,149.511
C09768=1127.185,405.482,-90.654,-176.768,11.508,149.512
C09769=1127.181,405.730,-90.692,-176.768,11.512,149.513
C09770=1127.177,405.976,-90.730,-176.768,11.516,149.514
C09771=1127.174,406.223,-90.768,-176.768,11.520,149.515
C09772=1127.170,406.471,-90.807,-176.767,11.524,149.516
C09773=1127.166,406.717,-90.844,-176.768,11.528,149.517
C09774=1127.163,406.964,-90.884,-176.767,11.531,149.518
C09775=1127.160,407.211,-90.922,-176.767,11.535,149.519
C09776=1127.155,407.458,-90.960,-176.767,11.539,149.520
C09777=1127.152,407.705,-90.998,-176.767,11.543,149.521
C09778=1127.148,407.953,-91.037,-176.768,11.547,149.522
C09779=1127.145,408.200,-91.075,-176.768,11.551,149.523
C09780=1127.141,408.446,-91.114,-176.768,11.555,149.524
C09781=1127.138,408.693,-91.152,-176.767,11.560,149.525
C09782=1127.134,408.941,-91.190,-176.767,11.564,149.526
C09783=1127.130,409.187,-91.229,-176.768,11.568,149.528
C09784=1127.126,409.434,-91.267,-176.768,11.572,149.529
C09785=1127.123,409.681,-91.306,-176.768,11.577,149.530
C09786=1127.120,409.929,-91.344,-176.768,11.581,149.531
C09787=1127.115,410.176,-91.383,-176.769,11.585,149.532
C09788=1127.112,410.422,-91.421,-176.769,11.589,149.533
C09789=1127.108,410.670,-91.460,-176.769,11.594,149.535
C09790=1127.105,410.916,-91.498,-176.769,11.598,149.536
C09791=1127.101,411.163,-91.537,-176.770,11.603,149.537
C09792=1127.097,411.410,-91.576,-176.770,11.607,149.538
C09793=1127.094,411.658,-91.614,-176.770,11.612,149.540
C09794=1127.090,411.904,-91.653,-176.770,11.617,149.541
C09795=1127.087,412.151,-91.691,-176.771,11.621,149.542
C09796=1127.083,412.398,-91.730,-176.771,11.625,149.543
C09797=1127.079,412.646,-91.768,-176.771,11.630,149.545
C09798=1127.076,412.892,-91.807,-176.772,11.635,149.546
C09799=1127.072,413.139,-91.845,-176.772,11.639,149.547
C09800=1127.068,413.386,-91.884,-176.773,11.644,149.549
C09801=1127.065,413.633,-91.922,-176.773,11.649,149.550
C09802=1127.061,413.880,-91.961,-176.774,11.654,149.551
C09803=1127.057,414.127,-91.999,-176.774,11.659,149.553
C09804=1127.055,414.374,-92.038,-176.775,11.664,149.554
C09805=1127.052,414.621,-92.077,-176.776,11.668,149.556
C09806=1127.051,414.868,-92.115,-176.776,11.674,149.557
C09807=1127.050,415.115,-92.153,-176.777,11.678,149.559
C09808=1127.050,415.362,-92.191,-176.777,11.683,149.560
C09809=1127.049,415.610,-92.229,-176.778,11.689,149.561
C09810=1127.050,415.821,-92.262,-176.778,11.693,149.563
C09811=1127.052,416.034,-92.294,-176.780,11.697,149.564
C09812=1127.052,416.245,-92.327,-176.780,11.701,149.565
C09813=1127.054,416.458,-92.359,-176.781,11.706,149.567
C09814=1127.056,416.670,-92.392,-176.781,11.710,149.568
C09815=1127.060,416.882,-92.424,-176.782,11.715,149.569
C09816=1127.063,417.094,-92.457,-176.783,11.719,149.571
C09817=1127.066,417.307,-92.489,-176.783,11.724,149.572
C09818=1126.647,417.306,-92.552,-176.776,11.728,149.571
C09819=1126.643,417.094,-92.519,-176.775,11.723,149.570
C09820=1126.641,416.882,-92.487,-176.775,11.719,149.569
C09821=1126.637,416.670,-92.454,-176.774,11.714,149.567
C09822=1126.635,416.458,-92.422,-176.773,11.710,149.566
C09823=1126.633,416.245,-92.390,-176.773,11.705,149.565
C09824=1126.632,416.033,-92.357,-176.772,11.701,149.563
C09825=1126.631,415.822,-92.324,-176.772,11.697,149.562
C09826=1126.631,415.610,-92.292,-176.771,11.692,149.561
C09827=1126.631,415.362,-92.254,-176.770,11.687,149.559
C09828=1126.631,415.115,-92.215,-176.769,11.683,149.558
C09829=1126.631,414.869,-92.177,-176.769,11.677,149.556
C09830=1126.633,414.622,-92.139,-176.768,11.673,149.555
C09831=1126.636,414.374,-92.101,-176.768,11.667,149.553
C09832=1126.638,414.127,-92.062,-176.767,11.663,149.552
C09833=1126.641,413.880,-92.023,-176.767,11.657,149.551
C09834=1126.645,413.633,-91.985,-176.767,11.653,149.549
C09835=1126.648,413.386,-91.946,-176.766,11.649,149.548
C09836=1126.653,413.139,-91.908,-176.766,11.643,149.547
C09837=1126.656,412.892,-91.869,-176.765,11.639,149.545
C09838=1126.659,412.645,-91.831,-176.765,11.634,149.544
C09839=1126.663,412.398,-91.791,-176.765,11.629,149.543
C09840=1126.668,412.151,-91.753,-176.764,11.625,149.541
C09841=1126.670,411.904,-91.715,-176.764,11.620,149.540
C09842=1126.674,411.657,-91.676,-176.764,11.615,149.539
C09843=1126.677,411.410,-91.637,-176.764,11.611,149.538
C09844=1126.682,411.163,-91.599,-176.763,11.607,149.536
C09845=1126.685,410.916,-91.560,-176.763,11.602,149.535
C09846=1126.689,410.669,-91.522,-176.763,11.597,149.534
C09847=1126.692,410.422,-91.483,-176.763,11.593,149.533
C09848=1126.696,410.176,-91.445,-176.762,11.589,149.532
C09849=1126.700,409.929,-91.406,-176.763,11.584,149.530
C09850=1126.704,409.681,-91.367,-176.762,11.580,149.529
C09851=1126.706,409.434,-91.329,-176.762,11.576,149.528
C09852=1126.711,409.188,-91.291,-176.762,11.571,149.527
C09853=1126.714,408.940,-91.253,-176.762,11.567,149.526
C09854=1126.718,408.693,-91.213,-176.762,11.563,149.525
C09855=1126.722,408.447,-91.176,-176.762,11.559,149.524
C09856=1126.725,408.200,-91.137,-176.762,11.555,149.523
C09857=1126.729,407.952,-91.098,-176.762,11.551,149.522
C09858=1126.732,407.705,-91.060,-176.762,11.547,149.521
C09859=1126.737,407.459,-91.021,-176.762,11.543,149.519
C09860=1126.740,407.211,-90.983,-176.762,11.539,149.518
C09861=1126.743,406.964,-90.944,-176.762,11.535,149.517
C09862=1126.747,406.718,-90.906,-176.762,11.531,149.516
C09863=1126.751,406.470,-90.868,-176.763,11.526,149.515
C09864=1126.754,406.224,-90.829,-176.763,11.523,149.515
C09865=1126.758,405.976,-90.791,-176.763,11.519,149.513
C09866=1126.762,405.729,-90.753,-176.763,11.515,149.513
C09867=1126.766,405.482,-90.715,-176.763,11.511,149.512
C09868=1126.768,405.235,-90.676,-176.764,11.507,149.511
C09869=1126.773,404.988,-90.638,-176.764,11.504,149.510
C09870=1126.776,404.741,-90.600,-176.764,11.500,149.509
C09871=1126.780,404.494,-90.561,-176.765,11.496,149.508
C09872=1126.784,404.248,-90.523,-176.765,11.493,149.507
C09873=1126.788,404.000,-90.485,-176.765,11.489,149.506
C09874=1126.791,403.753,-90.447,-176.765,11.485,149.505
C09875=1126.794,403.541,-90.413,-176.766,11.483,149.505
C09876=1126.797,403.329,-90.381,-176.766,11.479,149.504
C09877=1126.801,403.117,-90.347,-176.766,11.477,149.503
C09878=1126.803,402.904,-90.314,-176.767,11.473,149.503
C09879=1126.807,402.692,-90.282,-176.767,11.471,149.502
C09880=1126.809,402.480,-90.249,-176.767,11.467,149.501
C09881=1126.813,402.268,-90.217,-176.767,11.465,149.501
C09882=1126.816,402.055,-90.184,-176.768,11.461,149.500
C09883=1126.820,401.808,-90.145,-176.768,11.459,149.499
C09884=1126.823,401.561,-90.107,-176.769,11.455,149.498
C09885=1126.827,401.315,-90.069,-176.769,11.452,149.498
C09886=1126.831,401.067,-90.031,-176.770,11.448,149.497
C09887=1126.834,400.820,-89.993,-176.770,11.445,149.496
C09888=1126.838,400.574,-89.954,-176.771,11.442,149.495
C09889=1126.841,400.326,-89.916,-176.772,11.438,149.495
C09890=1126.846,400.079,-89.878,-176.772,11.436,149.494
C09891=1126.849,399.832,-89.840,-176.772,11.432,149.493
C09892=1126.852,399.585,-89.802,-176.773,11.429,149.493
C09893=1126.857,399.338,-89.764,-176.774,11.426,149.492
C09894=1126.860,399.091,-89.726,-176.775,11.423,149.491
C09895=1126.864,398.843,-89.687,-176.775,11.420,149.491
C09896=1126.867,398.597,-89.649,-176.776,11.417,149.490
C09897=1126.871,398.350,-89.611,-176.777,11.414,149.490
C09898=1126.875,398.103,-89.573,-176.777,11.410,149.489
C09899=1126.878,397.856,-89.535,-176.778,11.408,149.488
C09900=1126.881,397.608,-89.497,-176.779,11.405,149.488
C09901=1126.886,397.362,-89.459,-176.780,11.402,149.487
C09902=1126.889,397.114,-89.421,-176.780,11.400,149.487
C09903=1126.894,396.867,-89.383,-176.781,11.396,149.486
C09904=1126.897,396.620,-89.345,-176.782,11.393,149.486
C09905=1126.901,396.374,-89.307,-176.783,11.390,149.485
C09906=1126.905,396.126,-89.269,-176.784,11.388,149.485
C09907=1126.908,395.879,-89.231,-176.785,11.385,149.484
C09908=1126.912,395.632,-89.193,-176.786,11.382,149.484
C09909=1126.916,395.385,-89.155,-176.786,11.380,149.483
C09910=1126.919,395.138,-89.117,-176.787,11.377,149.483
C09911=1126.922,394.891,-89.079,-176.788,11.374,149.482
C09912=1126.927,394.644,-89.041,-176.789,11.371,149.482
C09913=1126.930,394.397,-89.003,-176.790,11.368,149.481
C09914=1126.933,394.149,-88.965,-176.791,11.367,149.481
C09915=1126.938,393.902,-88.927,-176.792,11.364,149.480
C09916=1126.941,393.655,-88.889,-176.793,11.361,149.480
C09917=1126.945,393.409,-88.851,-176.794,11.359,149.480
C09918=1126.948,393.161,-88.813,-176.795,11.356,149.479
C09919=1126.953,392.914,-88.775,-176.796,11.354,149.479
C09920=1126.956,392.667,-88.737,-176.797,11.351,149.479
C09921=1126.960,392.421,-88.700,-176.798,11.348,149.478
C09922=1126.964,392.172,-88.662,-176.799,11.346,149.478
C09923=1126.968,391.926,-88.624,-176.801,11.343,149.477
C09924=1126.971,391.679,-88.586,-176.802,11.341,149.477
C09925=1126.975,391.432,-88.549,-176.803,11.339,149.477
C09926=1126.978,391.185,-88.511,-176.803,11.337,149.476
C09927=1126.982,390.937,-88.472,-176.805,11.334,149.476
C09928=1126.985,390.691,-88.435,-176.806,11.332,149.476
C09929=1126.989,390.443,-88.397,-176.807,11.329,149.475
C09930=1126.993,390.196,-88.360,-176.809,11.327,149.475
C09931=1126.996,389.984,-88.327,-176.810,11.325,149.475
C09932=1127.000,389.771,-88.295,-176.811,11.323,149.475
C09933=1127.002,389.559,-88.263,-176.812,11.321,149.474
C09934=1127.005,389.346,-88.230,-176.813,11.320,149.474
C09935=1127.009,389.134,-88.197,-176.814,11.318,149.474
C09936=1127.012,388.922,-88.165,-176.815,11.316,149.474
C09937=1127.015,388.710,-88.133,-176.817,11.314,149.474
C09938=1127.018,388.497,-88.100,-176.818,11.312,149.474
C09939=1127.022,388.250,-88.062,-176.819,11.310,149.473
C09940=1127.025,388.003,-88.025,-176.820,11.307,149.473
C09941=1127.029,387.756,-87.987,-176.821,11.306,149.473
C09942=1127.033,387.509,-87.949,-176.823,11.303,149.473
C09943=1127.037,387.261,-87.911,-176.824,11.302,149.473
C09944=1127.040,387.015,-87.874,-176.825,11.300,149.472
C09945=1127.044,386.767,-87.836,-176.827,11.298,149.472
C09946=1127.048,386.520,-87.799,-176.828,11.296,149.472
C09947=1127.052,386.274,-87.761,-176.830,11.293,149.472
C09948=1127.055,386.026,-87.723,-176.831,11.292,149.472
C09949=1127.060,385.779,-87.686,-176.833,11.289,149.472
C09950=1127.063,385.532,-87.648,-176.834,11.288,149.472
C09951=1127.067,385.285,-87.610,-176.836,11.285,149.471
C09952=1127.070,385.037,-87.573,-176.837,11.284,149.471
C09953=1127.074,384.791,-87.536,-176.839,11.282,149.471
C09954=1127.077,384.543,-87.498,-176.841,11.280,149.471
C09955=1127.081,384.296,-87.461,-176.842,11.278,149.471
C09956=1127.085,384.049,-87.422,-176.844,11.276,149.471
C09957=1127.089,383.802,-87.385,-176.845,11.274,149.471
C09958=1127.093,383.555,-87.348,-176.847,11.273,149.471
C09959=1127.096,383.308,-87.310,-176.849,11.271,149.471
C09960=1127.100,383.060,-87.273,-176.851,11.268,149.471
C09961=1127.103,382.813,-87.235,-176.855,11.266,149.471
C09962=1127.107,382.567,-87.198,-176.857,11.264,149.471
C09963=1127.111,382.319,-87.161,-176.860,11.261,149.471
C09964=1127.114,382.072,-87.123,-176.862,11.259,149.471
C09965=1127.119,381.825,-87.086,-176.865,11.256,149.471
C09966=1127.122,381.578,-87.048,-176.868,11.253,149.471
C09967=1127.126,381.330,-87.011,-176.871,11.251,149.471
C09968=1127.130,381.084,-86.974,-176.874,11.249,149.472
C09969=1127.133,380.836,-86.936,-176.876,11.247,149.472
C09970=1127.137,380.589,-86.899,-176.879,11.244,149.472
C09971=1127.140,380.342,-86.861,-176.882,11.242,149.472
C09972=1127.144,380.095,-86.824,-176.885,11.240,149.472
C09973=1127.148,379.848,-86.787,-176.888,11.237,149.472
C09974=1127.152,379.600,-86.750,-176.891,11.234,149.472
C09975=1127.156,379.353,-86.712,-176.893,11.232,149.472
C09976=1127.160,379.106,-86.675,-176.896,11.230,149.472
C09977=1127.163,378.859,-86.637,-176.899,11.227,149.472
C09978=1127.167,378.612,-86.601,-176.902,11.225,149.473
C09979=1127.171,378.365,-86.564,-176.905,11.223,149.473
C09980=1127.174,378.117,-86.526,-176.908,11.220,149.473
C09981=1127.178,377.870,-86.489,-176.911,11.218,149.473
C09982=1127.182,377.623,-86.452,-176.914,11.215,149.473
C09983=1127.186,377.376,-86.414,-176.916,11.214,149.473
C09984=1127.190,377.128,-86.377,-176.919,11.211,149.473
C09985=1127.194,376.881,-86.340,-176.923,11.208,149.474
C09986=1127.198,376.634,-86.304,-176.926,11.206,149.474
C09987=1127.201,376.422,-86.272,-176.928,11.204,149.474
C09988=1127.204,376.209,-86.240,-176.931,11.202,149.474
C09989=1127.207,375.997,-86.208,-176.933,11.200,149.474
C09990=1127.210,375.784,-86.176,-176.935,11.198,149.474
C09991=1127.214,375.572,-86.144,-176.938,11.196,149.474
C09992=1127.217,375.359,-86.113,-176.941,11.194,149.474
C09993=1127.220,375.147,-86.081,-176.944,11.192,149.475
C09994=1127.223,374.934,-86.049,-176.946,11.190,149.475
C09995=1127.227,374.687,-86.012,-176.949,11.187,149.475
C09996=1127.230,374.440,-85.975,-176.952,11.186,149.475
//INST
///DATE 2021/06/25 14:32
///ATTR SC,RW,RJ
////FRAME ROBOT
///GROUP1 RB1
NOP
MOVL C00000 V=800.0 PL=0
MOVL C00001 V=800.0 PL=0
MOVL C00002 V=800.0 PL=0
MOVL C00003 V=800.0 PL=0
MOVL C00004 V=800.0 PL=0
MOVL C00005 V=800.0 PL=0
MOVL C00006 V=800.0 PL=0
MOVL C00007 V=800.0 PL=0
MOVL C00008 V=800.0 PL=0
MOVL C00009 V=800.0 PL=0
MOVL C00010 V=800.0 PL=0
MOVL C00011 V=800.0 PL=0
MOVL C00012 V=800.0 PL=0
MOVL C00013 V=800.0 PL=0
MOVL C00014 V=800.0 PL=0
MOVL C00015 V=800.0 PL=0
MOVL C00016 V=800.0 PL=0
MOVL C00017 V=800.0 PL=0
MOVL C00018 V=800.0 PL=0
MOVL C00019 V=800.0 PL=0
MOVL C00020 V=800.0 PL=0
MOVL C00021 V=800.0 PL=0
MOVL C00022 V=800.0 PL=0
MOVL C00023 V=800.0 PL=0
MOVL C00024 V=800.0 PL=0
MOVL C00025 V=800.0 PL=0
MOVL C00026 V=800.0 PL=0
MOVL C00027 V=800.0 PL=0
MOVL C00028 V=800.0 PL=0
MOVL C00029 V=800.0 PL=0
MOVL C00030 V=800.0 PL=0
MOVL C00031 V=800.0 PL=0
MOVL C00032 V=800.0 PL=0
MOVL C00033 V=800.0 PL=0
MOVL C00034 V=800.0 PL=0
MOVL C00035 V=800.0 PL=0
MOVL C00036 V=800.0 PL=0
MOVL C00037 V=800.0 PL=0
MOVL C00038 V=800.0 PL=0
MOVL C00039 V=800.0 PL=0
MOVL C00040 V=800.0 PL=0
MOVL C00041 V=800.0 PL=0
MOVL C00042 V=800.0 PL=0
MOVL C00043 V=800.0 PL=0
MOVL C00044 V=800.0 PL=0
MOVL C00045 V=800.0 PL=0
MOVL C00046 V=800.0 PL=0
MOVL C00047 V=800.0 PL=0
MOVL C00048 V=800.0 PL=0
MOVL C00049 V=800.0 PL=0
MOVL C00050 V=800.0 PL=0
MOVL C00051 V=800.0 PL=0
MOVL C00052 V=800.0 PL=0
MOVL C00053 V=800.0 PL=0
MOVL C00054 V=800.0 PL=0
MOVL C00055 V=800.0 PL=0
MOVL C00056 V=800.0 PL=0
MOVL C00057 V=800.0 PL=0
MOVL C00058 V=800.0 PL=0
MOVL C00059 V=800.0 PL=0
MOVL C00060 V=800.0 PL=0
MOVL C00061 V=800.0 PL=0
MOVL C00062 V=800.0 PL=0
MOVL C00063 V=800.0 PL=0
MOVL C00064 V=800.0 PL=0
MOVL C00065 V=800.0 PL=0
MOVL C00066 V=800.0 PL=0
MOVL C00067 V=800.0 PL=0
MOVL C00068 V=800.0 PL=0
MOVL C00069 V=800.0 PL=0
MOVL C00070 V=800.0 PL=0
MOVL C00071 V=800.0 PL=0
MOVL C00072 V=800.0 PL=0
MOVL C00073 V=800.0 PL=0
MOVL C00074 V=800.0 PL=0
MOVL C00075 V=800.0 PL=0
MOVL C00076 V=800.0 PL=0
MOVL C00077 V=800.0 PL=0
MOVL C00078 V=800.0 PL=0
MOVL C00079 V=800.0 PL=0
MOVL C00080 V=800.0 PL=0
MOVL C00081 V=800.0 PL=0
MOVL C00082 V=800.0 PL=0
MOVL C00083 V=800.0 PL=0
MOVL C00084 V=800.0 PL=0
MOVL C00085 V=800.0 PL=0
MOVL C00086 V=800.0 PL=0
MOVL C00087 V=800.0 PL=0
MOVL C00088 V=800.0 PL=0
MOVL C00089 V=800.0 PL=0
MOVL C00090 V=800.0 PL=0
MOVL C00091 V=800.0 PL=0
MOVL C00092 V=800.0 PL=0
MOVL C00093 V=800.0 PL=0
MOVL C00094 V=800.0 PL=0
MOVL C00095 V=800.0 PL=0
MOVL C00096 V=800.0 PL=0
MOVL C00097 V=800.0 PL=0
MOVL C00098 V=800.0 PL=0
MOVL C00099 V=800.0 PL=0
MOVL C00100 V=800.0 PL=0
MOVL C00101 V=800.0 PL=0
MOVL C00102 V=800.0 PL=0
MOVL C00103 V=800.0 PL=0
MOVL C00104 V=800.0 PL=0
MOVL C00105 V=800.0 PL=0
MOVL C00106 V=800.0 PL=0
MOVL C00107 V=800.0 PL=0
MOVL C00108 V=800.0 PL=0
MOVL C00109 V=800.0 PL=0
MOVL C00110 V=800.0 PL=0
MOVL C00111 V=800.0 PL=0
MOVL C00112 V=800.0 PL=0
MOVL C00113 V=800.0 PL=0
MOVL C00114 V=800.0 PL=0
MOVL C00115 V=800.0 PL=0
MOVL C00116 V=800.0 PL=0
MOVL C00117 V=800.0 PL=0
MOVL C00118 V=800.0 PL=0
MOVL C00119 V=800.0 PL=0
MOVL C00120 V=800.0 PL=0
MOVL C00121 V=800.0 PL=0
MOVL C00122 V=800.0 PL=0
MOVL C00123 V=800.0 PL=0
MOVL C00124 V=800.0 PL=0
MOVL C00125 V=800.0 PL=0
MOVL C00126 V=800.0 PL=0
MOVL C00127 V=800.0 PL=0
MOVL C00128 V=800.0 PL=0
MOVL C00129 V=800.0 PL=0
MOVL C00130 V=800.0 PL=0
MOVL C00131 V=800.0 PL=0
MOVL C00132 V=800.0 PL=0
MOVL C00133 V=800.0 PL=0
MOVL C00134 V=800.0 PL=0
MOVL C00135 V=800.0 PL=0
MOVL C00136 V=800.0 PL=0
MOVL C00137 V=800.0 PL=0
MOVL C00138 V=800.0 PL=0
MOVL C00139 V=800.0 PL=0
MOVL C00140 V=800.0 PL=0
MOVL C00141 V=800.0 PL=0
MOVL C00142 V=800.0 PL=0
MOVL C00143 V=800.0 PL=0
MOVL C00144 V=800.0 PL=0
MOVL C00145 V=800.0 PL=0
MOVL C00146 V=800.0 PL=0
MOVL C00147 V=800.0 PL=0
MOVL C00148 V=800.0 PL=0
MOVL C00149 V=800.0 PL=0
MOVL C00150 V=800.0 PL=0
MOVL C00151 V=800.0 PL=0
MOVL C00152 V=800.0 PL=0
MOVL C00153 V=800.0 PL=0
MOVL C00154 V=800.0 PL=0
MOVL C00155 V=800.0 PL=0
MOVL C00156 V=800.0 PL=0
MOVL C00157 V=800.0 PL=0
MOVL C00158 V=800.0 PL=0
MOVL C00159 V=800.0 PL=0
MOVL C00160 V=800.0 PL=0
MOVL C00161 V=800.0 PL=0
MOVL C00162 V=800.0 PL=0
MOVL C00163 V=800.0 PL=0
MOVL C00164 V=800.0 PL=0
MOVL C00165 V=800.0 PL=0
MOVL C00166 V=800.0 PL=0
MOVL C00167 V=800.0 PL=0
MOVL C00168 V=800.0 PL=0
MOVL C00169 V=800.0 PL=0
MOVL C00170 V=800.0 PL=0
MOVL C00171 V=800.0 PL=0
MOVL C00172 V=800.0 PL=0
MOVL C00173 V=800.0 PL=0
MOVL C00174 V=800.0 PL=0
MOVL C00175 V=800.0 PL=0
MOVL C00176 V=800.0 PL=0
MOVL C00177 V=800.0 PL=0
MOVL C00178 V=800.0 PL=0
MOVL C00179 V=800.0 PL=0
MOVL C00180 V=800.0 PL=0
MOVL C00181 V=800.0 PL=0
MOVL C00182 V=800.0 PL=0
MOVL C00183 V=800.0 PL=0
MOVL C00184 V=800.0 PL=0
MOVL C00185 V=800.0 PL=0
MOVL C00186 V=800.0 PL=0
MOVL C00187 V=800.0 PL=0
MOVL C00188 V=800.0 PL=0
MOVL C00189 V=800.0 PL=0
MOVL C00190 V=800.0 PL=0
MOVL C00191 V=800.0 PL=0
MOVL C00192 V=800.0 PL=0
MOVL C00193 V=800.0 PL=0
MOVL C00194 V=800.0 PL=0
MOVL C00195 V=800.0 PL=0
MOVL C00196 V=800.0 PL=0
MOVL C00197 V=800.0 PL=0
MOVL C00198 V=800.0 PL=0
MOVL C00199 V=800.0 PL=0
MOVL C00200 V=800.0 PL=0
MOVL C00201 V=800.0 PL=0
MOVL C00202 V=800.0 PL=0
MOVL C00203 V=800.0 PL=0
MOVL C00204 V=800.0 PL=0
MOVL C00205 V=800.0 PL=0
MOVL C00206 V=800.0 PL=0
MOVL C00207 V=800.0 PL=0
MOVL C00208 V=800.0 PL=0
MOVL C00209 V=800.0 PL=0
MOVL C00210 V=800.0 PL=0
MOVL C00211 V=800.0 PL=0
MOVL C00212 V=800.0 PL=0
MOVL C00213 V=800.0 PL=0
MOVL C00214 V=800.0 PL=0
MOVL C00215 V=800.0 PL=0
MOVL C00216 V=800.0 PL=0
MOVL C00217 V=800.0 PL=0
MOVL C00218 V=800.0 PL=0
MOVL C00219 V=800.0 PL=0
MOVL C00220 V=800.0 PL=0
MOVL C00221 V=800.0 PL=0
MOVL C00222 V=800.0 PL=0
MOVL C00223 V=800.0 PL=0
MOVL C00224 V=800.0 PL=0
MOVL C00225 V=800.0 PL=0
MOVL C00226 V=800.0 PL=0
MOVL C00227 V=800.0 PL=0
MOVL C00228 V=800.0 PL=0
MOVL C00229 V=800.0 PL=0
MOVL C00230 V=800.0 PL=0
MOVL C00231 V=800.0 PL=0
MOVL C00232 V=800.0 PL=0
MOVL C00233 V=800.0 PL=0
MOVL C00234 V=800.0 PL=0
MOVL C00235 V=800.0 PL=0
MOVL C00236 V=800.0 PL=0
MOVL C00237 V=800.0 PL=0
MOVL C00238 V=800.0 PL=0
MOVL C00239 V=800.0 PL=0
MOVL C00240 V=800.0 PL=0
MOVL C00241 V=800.0 PL=0
MOVL C00242 V=800.0 PL=0
MOVL C00243 V=800.0 PL=0
MOVL C00244 V=800.0 PL=0
MOVL C00245 V=800.0 PL=0
MOVL C00246 V=800.0 PL=0
MOVL C00247 V=800.0 PL=0
MOVL C00248 V=800.0 PL=0
MOVL C00249 V=800.0 PL=0
MOVL C00250 V=800.0 PL=0
MOVL C00251 V=800.0 PL=0
MOVL C00252 V=800.0 PL=0
MOVL C00253 V=800.0 PL=0
MOVL C00254 V=800.0 PL=0
MOVL C00255 V=800.0 PL=0
MOVL C00256 V=800.0 PL=0
MOVL C00257 V=800.0 PL=0
MOVL C00258 V=800.0 PL=0
MOVL C00259 V=800.0 PL=0
MOVL C00260 V=800.0 PL=0
MOVL C00261 V=800.0 PL=0
MOVL C00262 V=800.0 PL=0
MOVL C00263 V=800.0 PL=0
MOVL C00264 V=800.0 PL=0
MOVL C00265 V=800.0 PL=0
MOVL C00266 V=800.0 PL=0
MOVL C00267 V=800.0 PL=0
MOVL C00268 V=800.0 PL=0
MOVL C00269 V=800.0 PL=0
MOVL C00270 V=800.0 PL=0
MOVL C00271 V=800.0 PL=0
MOVL C00272 V=800.0 PL=0
MOVL C00273 V=800.0 PL=0
MOVL C00274 V=800.0 PL=0
MOVL C00275 V=800.0 PL=0
MOVL C00276 V=800.0 PL=0
MOVL C00277 V=800.0 PL=0
MOVL C00278 V=800.0 PL=0
MOVL C00279 V=800.0 PL=0
MOVL C00280 V=800.0 PL=0
MOVL C00281 V=800.0 PL=0
MOVL C00282 V=800.0 PL=0
MOVL C00283 V=800.0 PL=0
MOVL C00284 V=800.0 PL=0
MOVL C00285 V=800.0 PL=0
MOVL C00286 V=800.0 PL=0
MOVL C00287 V=800.0 PL=0
MOVL C00288 V=800.0 PL=0
MOVL C00289 V=800.0 PL=0
MOVL C00290 V=800.0 PL=0
MOVL C00291 V=800.0 PL=0
MOVL C00292 V=800.0 PL=0
MOVL C00293 V=800.0 PL=0
MOVL C00294 V=800.0 PL=0
MOVL C00295 V=800.0 PL=0
MOVL C00296 V=800.0 PL=0
MOVL C00297 V=800.0 PL=0
MOVL C00298 V=800.0 PL=0
MOVL C00299 V=800.0 PL=0
MOVL C00300 V=800.0 PL=0
MOVL C00301 V=800.0 PL=0
MOVL C00302 V=800.0 PL=0
MOVL C00303 V=800.0 PL=0
MOVL C00304 V=800.0 PL=0
MOVL C00305 V=800.0 PL=0
MOVL C00306 V=800.0 PL=0
MOVL C00307 V=800.0 PL=0
MOVL C00308 V=800.0 PL=0
MOVL C00309 V=800.0 PL=0
MOVL C00310 V=800.0 PL=0
MOVL C00311 V=800.0 PL=0
MOVL C00312 V=800.0 PL=0
MOVL C00313 V=800.0 PL=0
MOVL C00314 V=800.0 PL=0
MOVL C00315 V=800.0 PL=0
MOVL C00316 V=800.0 PL=0
MOVL C00317 V=800.0 PL=0
MOVL C00318 V=800.0 PL=0
MOVL C00319 V=800.0 PL=0
MOVL C00320 V=800.0 PL=0
MOVL C00321 V=800.0 PL=0
MOVL C00322 V=800.0 PL=0
MOVL C00323 V=800.0 PL=0
MOVL C00324 V=800.0 PL=0
MOVL C00325 V=800.0 PL=0
MOVL C00326 V=800.0 PL=0
MOVL C00327 V=800.0 PL=0
MOVL C00328 V=800.0 PL=0
MOVL C00329 V=800.0 PL=0
MOVL C00330 V=800.0 PL=0
MOVL C00331 V=800.0 PL=0
MOVL C00332 V=800.0 PL=0
MOVL C00333 V=800.0 PL=0
MOVL C00334 V=800.0 PL=0
MOVL C00335 V=800.0 PL=0
MOVL C00336 V=800.0 PL=0
MOVL C00337 V=800.0 PL=0
MOVL C00338 V=800.0 PL=0
MOVL C00339 V=800.0 PL=0
MOVL C00340 V=800.0 PL=0
MOVL C00341 V=800.0 PL=0
MOVL C00342 V=800.0 PL=0
MOVL C00343 V=800.0 PL=0
MOVL C00344 V=800.0 PL=0
MOVL C00345 V=800.0 PL=0
MOVL C00346 V=800.0 PL=0
MOVL C00347 V=800.0 PL=0
MOVL C00348 V=800.0 PL=0
MOVL C00349 V=800.0 PL=0
MOVL C00350 V=800.0 PL=0
MOVL C00351 V=800.0 PL=0
MOVL C00352 V=800.0 PL=0
MOVL C00353 V=800.0 PL=0
MOVL C00354 V=800.0 PL=0
MOVL C00355 V=800.0 PL=0
MOVL C00356 V=800.0 PL=0
MOVL C00357 V=800.0 PL=0
MOVL C00358 V=800.0 PL=0
MOVL C00359 V=800.0 PL=0
MOVL C00360 V=800.0 PL=0
MOVL C00361 V=800.0 PL=0
MOVL C00362 V=800.0 PL=0
MOVL C00363 V=800.0 PL=0
MOVL C00364 V=800.0 PL=0
MOVL C00365 V=800.0 PL=0
MOVL C00366 V=800.0 PL=0
MOVL C00367 V=800.0 PL=0
MOVL C00368 V=800.0 PL=0
MOVL C00369 V=800.0 PL=0
MOVL C00370 V=800.0 PL=0
MOVL C00371 V=800.0 PL=0
MOVL C00372 V=800.0 PL=0
MOVL C00373 V=800.0 PL=0
MOVL C00374 V=800.0 PL=0
MOVL C00375 V=800.0 PL=0
MOVL C00376 V=800.0 PL=0
MOVL C00377 V=800.0 PL=0
MOVL C00378 V=800.0 PL=0
MOVL C00379 V=800.0 PL=0
MOVL C00380 V=800.0 PL=0
MOVL C00381 V=800.0 PL=0
MOVL C00382 V=800.0 PL=0
MOVL C00383 V=800.0 PL=0
MOVL C00384 V=800.0 PL=0
MOVL C00385 V=800.0 PL=0
MOVL C00386 V=800.0 PL=0
MOVL C00387 V=800.0 PL=0
MOVL C00388 V=800.0 PL=0
MOVL C00389 V=800.0 PL=0
MOVL C00390 V=800.0 PL=0
MOVL C00391 V=800.0 PL=0
MOVL C00392 V=800.0 PL=0
MOVL C00393 V=800.0 PL=0
MOVL C00394 V=800.0 PL=0
MOVL C00395 V=800.0 PL=0
MOVL C00396 V=800.0 PL=0
MOVL C00397 V=800.0 PL=0
MOVL C00398 V=800.0 PL=0
MOVL C00399 V=800.0 PL=0
MOVL C00400 V=800.0 PL=0
MOVL C00401 V=800.0 PL=0
MOVL C00402 V=800.0 PL=0
MOVL C00403 V=800.0 PL=0
MOVL C00404 V=800.0 PL=0
MOVL C00405 V=800.0 PL=0
MOVL C00406 V=800.0 PL=0
MOVL C00407 V=800.0 PL=0
MOVL C00408 V=800.0 PL=0
MOVL C00409 V=800.0 PL=0
MOVL C00410 V=800.0 PL=0
MOVL C00411 V=800.0 PL=0
MOVL C00412 V=800.0 PL=0
MOVL C00413 V=800.0 PL=0
MOVL C00414 V=800.0 PL=0
MOVL C00415 V=800.0 PL=0
MOVL C00416 V=800.0 PL=0
MOVL C00417 V=800.0 PL=0
MOVL C00418 V=800.0 PL=0
MOVL C00419 V=800.0 PL=0
MOVL C00420 V=800.0 PL=0
MOVL C00421 V=800.0 PL=0
MOVL C00422 V=800.0 PL=0
MOVL C00423 V=800.0 PL=0
MOVL C00424 V=800.0 PL=0
MOVL C00425 V=800.0 PL=0
MOVL C00426 V=800.0 PL=0
MOVL C00427 V=800.0 PL=0
MOVL C00428 V=800.0 PL=0
MOVL C00429 V=800.0 PL=0
MOVL C00430 V=800.0 PL=0
MOVL C00431 V=800.0 PL=0
MOVL C00432 V=800.0 PL=0
MOVL C00433 V=800.0 PL=0
MOVL C00434 V=800.0 PL=0
MOVL C00435 V=800.0 PL=0
MOVL C00436 V=800.0 PL=0
MOVL C00437 V=800.0 PL=0
MOVL C00438 V=800.0 PL=0
MOVL C00439 V=800.0 PL=0
MOVL C00440 V=800.0 PL=0
MOVL C00441 V=800.0 PL=0
MOVL C00442 V=800.0 PL=0
MOVL C00443 V=800.0 PL=0
MOVL C00444 V=800.0 PL=0
MOVL C00445 V=800.0 PL=0
MOVL C00446 V=800.0 PL=0
MOVL C00447 V=800.0 PL=0
MOVL C00448 V=800.0 PL=0
MOVL C00449 V=800.0 PL=0
MOVL C00450 V=800.0 PL=0
MOVL C00451 V=800.0 PL=0
MOVL C00452 V=800.0 PL=0
MOVL C00453 V=800.0 PL=0
MOVL C00454 V=800.0 PL=0
MOVL C00455 V=800.0 PL=0
MOVL C00456 V=800.0 PL=0
MOVL C00457 V=800.0 PL=0
MOVL C00458 V=800.0 PL=0
MOVL C00459 V=800.0 PL=0
MOVL C00460 V=800.0 PL=0
MOVL C00461 V=800.0 PL=0
MOVL C00462 V=800.0 PL=0
MOVL C00463 V=800.0 PL=0
MOVL C00464 V=800.0 PL=0
MOVL C00465 V=800.0 PL=0
MOVL C00466 V=800.0 PL=0
MOVL C00467 V=800.0 PL=0
MOVL C00468 V=800.0 PL=0
MOVL C00469 V=800.0 PL=0
MOVL C00470 V=800.0 PL=0
MOVL C00471 V=800.0 PL=0
MOVL C00472 V=800.0 PL=0
MOVL C00473 V=800.0 PL=0
MOVL C00474 V=800.0 PL=0
MOVL C00475 V=800.0 PL=0
MOVL C00476 V=800.0 PL=0
MOVL C00477 V=800.0 PL=0
MOVL C00478 V=800.0 PL=0
MOVL C00479 V=800.0 PL=0
MOVL C00480 V=800.0 PL=0
MOVL C00481 V=800.0 PL=0
MOVL C00482 V=800.0 PL=0
MOVL C00483 V=800.0 PL=0
MOVL C00484 V=800.0 PL=0
MOVL C00485 V=800.0 PL=0
MOVL C00486 V=800.0 PL=0
MOVL C00487 V=800.0 PL=0
MOVL C00488 V=800.0 PL=0
MOVL C00489 V=800.0 PL=0
MOVL C00490 V=800.0 PL=0
MOVL C00491 V=800.0 PL=0
MOVL C00492 V=800.0 PL=0
MOVL C00493 V=800.0 PL=0
MOVL C00494 V=800.0 PL=0
MOVL C00495 V=800.0 PL=0
MOVL C00496 V=800.0 PL=0
MOVL C00497 V=800.0 PL=0
MOVL C00498 V=800.0 PL=0
MOVL C00499 V=800.0 PL=0
MOVL C00500 V=800.0 PL=0
MOVL C00501 V=800.0 PL=0
MOVL C00502 V=800.0 PL=0
MOVL C00503 V=800.0 PL=0
MOVL C00504 V=800.0 PL=0
MOVL C00505 V=800.0 PL=0
MOVL C00506 V=800.0 PL=0
MOVL C00507 V=800.0 PL=0
MOVL C00508 V=800.0 PL=0
MOVL C00509 V=800.0 PL=0
MOVL C00510 V=800.0 PL=0
MOVL C00511 V=800.0 PL=0
MOVL C00512 V=800.0 PL=0
MOVL C00513 V=800.0 PL=0
MOVL C00514 V=800.0 PL=0
MOVL C00515 V=800.0 PL=0
MOVL C00516 V=800.0 PL=0
MOVL C00517 V=800.0 PL=0
MOVL C00518 V=800.0 PL=0
MOVL C00519 V=800.0 PL=0
MOVL C00520 V=800.0 PL=0
MOVL C00521 V=800.0 PL=0
MOVL C00522 V=800.0 PL=0
MOVL C00523 V=800.0 PL=0
MOVL C00524 V=800.0 PL=0
MOVL C00525 V=800.0 PL=0
MOVL C00526 V=800.0 PL=0
MOVL C00527 V=800.0 PL=0
MOVL C00528 V=800.0 PL=0
MOVL C00529 V=800.0 PL=0
MOVL C00530 V=800.0 PL=0
MOVL C00531 V=800.0 PL=0
MOVL C00532 V=800.0 PL=0
MOVL C00533 V=800.0 PL=0
MOVL C00534 V=800.0 PL=0
MOVL C00535 V=800.0 PL=0
MOVL C00536 V=800.0 PL=0
MOVL C00537 V=800.0 PL=0
MOVL C00538 V=800.0 PL=0
MOVL C00539 V=800.0 PL=0
MOVL C00540 V=800.0 PL=0
MOVL C00541 V=800.0 PL=0
MOVL C00542 V=800.0 PL=0
MOVL C00543 V=800.0 PL=0
MOVL C00544 V=800.0 PL=0
MOVL C00545 V=800.0 PL=0
MOVL C00546 V=800.0 PL=0
MOVL C00547 V=800.0 PL=0
MOVL C00548 V=800.0 PL=0
MOVL C00549 V=800.0 PL=0
MOVL C00550 V=800.0 PL=0
MOVL C00551 V=800.0 PL=0
MOVL C00552 V=800.0 PL=0
MOVL C00553 V=800.0 PL=0
MOVL C00554 V=800.0 PL=0
MOVL C00555 V=800.0 PL=0
MOVL C00556 V=800.0 PL=0
MOVL C00557 V=800.0 PL=0
MOVL C00558 V=800.0 PL=0
MOVL C00559 V=800.0 PL=0
MOVL C00560 V=800.0 PL=0
MOVL C00561 V=800.0 PL=0
MOVL C00562 V=800.0 PL=0
MOVL C00563 V=800.0 PL=0
MOVL C00564 V=800.0 PL=0
MOVL C00565 V=800.0 PL=0
MOVL C00566 V=800.0 PL=0
MOVL C00567 V=800.0 PL=0
MOVL C00568 V=800.0 PL=0
MOVL C00569 V=800.0 PL=0
MOVL C00570 V=800.0 PL=0
MOVL C00571 V=800.0 PL=0
MOVL C00572 V=800.0 PL=0
MOVL C00573 V=800.0 PL=0
MOVL C00574 V=800.0 PL=0
MOVL C00575 V=800.0 PL=0
MOVL C00576 V=800.0 PL=0
MOVL C00577 V=800.0 PL=0
MOVL C00578 V=800.0 PL=0
MOVL C00579 V=800.0 PL=0
MOVL C00580 V=800.0 PL=0
MOVL C00581 V=800.0 PL=0
MOVL C00582 V=800.0 PL=0
MOVL C00583 V=800.0 PL=0
MOVL C00584 V=800.0 PL=0
MOVL C00585 V=800.0 PL=0
MOVL C00586 V=800.0 PL=0
MOVL C00587 V=800.0 PL=0
MOVL C00588 V=800.0 PL=0
MOVL C00589 V=800.0 PL=0
MOVL C00590 V=800.0 PL=0
MOVL C00591 V=800.0 PL=0
MOVL C00592 V=800.0 PL=0
MOVL C00593 V=800.0 PL=0
MOVL C00594 V=800.0 PL=0
MOVL C00595 V=800.0 PL=0
MOVL C00596 V=800.0 PL=0
MOVL C00597 V=800.0 PL=0
MOVL C00598 V=800.0 PL=0
MOVL C00599 V=800.0 PL=0
MOVL C00600 V=800.0 PL=0
MOVL C00601 V=800.0 PL=0
MOVL C00602 V=800.0 PL=0
MOVL C00603 V=800.0 PL=0
MOVL C00604 V=800.0 PL=0
MOVL C00605 V=800.0 PL=0
MOVL C00606 V=800.0 PL=0
MOVL C00607 V=800.0 PL=0
MOVL C00608 V=800.0 PL=0
MOVL C00609 V=800.0 PL=0
MOVL C00610 V=800.0 PL=0
MOVL C00611 V=800.0 PL=0
MOVL C00612 V=800.0 PL=0
MOVL C00613 V=800.0 PL=0
MOVL C00614 V=800.0 PL=0
MOVL C00615 V=800.0 PL=0
MOVL C00616 V=800.0 PL=0
MOVL C00617 V=800.0 PL=0
MOVL C00618 V=800.0 PL=0
MOVL C00619 V=800.0 PL=0
MOVL C00620 V=800.0 PL=0
MOVL C00621 V=800.0 PL=0
MOVL C00622 V=800.0 PL=0
MOVL C00623 V=800.0 PL=0
MOVL C00624 V=800.0 PL=0
MOVL C00625 V=800.0 PL=0
MOVL C00626 V=800.0 PL=0
MOVL C00627 V=800.0 PL=0
MOVL C00628 V=800.0 PL=0
MOVL C00629 V=800.0 PL=0
MOVL C00630 V=800.0 PL=0
MOVL C00631 V=800.0 PL=0
MOVL C00632 V=800.0 PL=0
MOVL C00633 V=800.0 PL=0
MOVL C00634 V=800.0 PL=0
MOVL C00635 V=800.0 PL=0
MOVL C00636 V=800.0 PL=0
MOVL C00637 V=800.0 PL=0
MOVL C00638 V=800.0 PL=0
MOVL C00639 V=800.0 PL=0
MOVL C00640 V=800.0 PL=0
MOVL C00641 V=800.0 PL=0
MOVL C00642 V=800.0 PL=0
MOVL C00643 V=800.0 PL=0
MOVL C00644 V=800.0 PL=0
MOVL C00645 V=800.0 PL=0
MOVL C00646 V=800.0 PL=0
MOVL C00647 V=800.0 PL=0
MOVL C00648 V=800.0 PL=0
MOVL C00649 V=800.0 PL=0
MOVL C00650 V=800.0 PL=0
MOVL C00651 V=800.0 PL=0
MOVL C00652 V=800.0 PL=0
MOVL C00653 V=800.0 PL=0
MOVL C00654 V=800.0 PL=0
MOVL C00655 V=800.0 PL=0
MOVL C00656 V=800.0 PL=0
MOVL C00657 V=800.0 PL=0
MOVL C00658 V=800.0 PL=0
MOVL C00659 V=800.0 PL=0
MOVL C00660 V=800.0 PL=0
MOVL C00661 V=800.0 PL=0
MOVL C00662 V=800.0 PL=0
MOVL C00663 V=800.0 PL=0
MOVL C00664 V=800.0 PL=0
MOVL C00665 V=800.0 PL=0
MOVL C00666 V=800.0 PL=0
MOVL C00667 V=800.0 PL=0
MOVL C00668 V=800.0 PL=0
MOVL C00669 V=800.0 PL=0
MOVL C00670 V=800.0 PL=0
MOVL C00671 V=800.0 PL=0
MOVL C00672 V=800.0 PL=0
MOVL C00673 V=800.0 PL=0
MOVL C00674 V=800.0 PL=0
MOVL C00675 V=800.0 PL=0
MOVL C00676 V=800.0 PL=0
MOVL C00677 V=800.0 PL=0
MOVL C00678 V=800.0 PL=0
MOVL C00679 V=800.0 PL=0
MOVL C00680 V=800.0 PL=0
MOVL C00681 V=800.0 PL=0
MOVL C00682 V=800.0 PL=0
MOVL C00683 V=800.0 PL=0
MOVL C00684 V=800.0 PL=0
MOVL C00685 V=800.0 PL=0
MOVL C00686 V=800.0 PL=0
MOVL C00687 V=800.0 PL=0
MOVL C00688 V=800.0 PL=0
MOVL C00689 V=800.0 PL=0
MOVL C00690 V=800.0 PL=0
MOVL C00691 V=800.0 PL=0
MOVL C00692 V=800.0 PL=0
MOVL C00693 V=800.0 PL=0
MOVL C00694 V=800.0 PL=0
MOVL C00695 V=800.0 PL=0
MOVL C00696 V=800.0 PL=0
MOVL C00697 V=800.0 PL=0
MOVL C00698 V=800.0 PL=0
MOVL C00699 V=800.0 PL=0
MOVL C00700 V=800.0 PL=0
MOVL C00701 V=800.0 PL=0
MOVL C00702 V=800.0 PL=0
MOVL C00703 V=800.0 PL=0
MOVL C00704 V=800.0 PL=0
MOVL C00705 V=800.0 PL=0
MOVL C00706 V=800.0 PL=0
MOVL C00707 V=800.0 PL=0
MOVL C00708 V=800.0 PL=0
MOVL C00709 V=800.0 PL=0
MOVL C00710 V=800.0 PL=0
MOVL C00711 V=800.0 PL=0
MOVL C00712 V=800.0 PL=0
MOVL C00713 V=800.0 PL=0
MOVL C00714 V=800.0 PL=0
MOVL C00715 V=800.0 PL=0
MOVL C00716 V=800.0 PL=0
MOVL C00717 V=800.0 PL=0
MOVL C00718 V=800.0 PL=0
MOVL C00719 V=800.0 PL=0
MOVL C00720 V=800.0 PL=0
MOVL C00721 V=800.0 PL=0
MOVL C00722 V=800.0 PL=0
MOVL C00723 V=800.0 PL=0
MOVL C00724 V=800.0 PL=0
MOVL C00725 V=800.0 PL=0
MOVL C00726 V=800.0 PL=0
MOVL C00727 V=800.0 PL=0
MOVL C00728 V=800.0 PL=0
MOVL C00729 V=800.0 PL=0
MOVL C00730 V=800.0 PL=0
MOVL C00731 V=800.0 PL=0
MOVL C00732 V=800.0 PL=0
MOVL C00733 V=800.0 PL=0
MOVL C00734 V=800.0 PL=0
MOVL C00735 V=800.0 PL=0
MOVL C00736 V=800.0 PL=0
MOVL C00737 V=800.0 PL=0
MOVL C00738 V=800.0 PL=0
MOVL C00739 V=800.0 PL=0
MOVL C00740 V=800.0 PL=0
MOVL C00741 V=800.0 PL=0
MOVL C00742 V=800.0 PL=0
MOVL C00743 V=800.0 PL=0
MOVL C00744 V=800.0 PL=0
MOVL C00745 V=800.0 PL=0
MOVL C00746 V=800.0 PL=0
MOVL C00747 V=800.0 PL=0
MOVL C00748 V=800.0 PL=0
MOVL C00749 V=800.0 PL=0
MOVL C00750 V=800.0 PL=0
MOVL C00751 V=800.0 PL=0
MOVL C00752 V=800.0 PL=0
MOVL C00753 V=800.0 PL=0
MOVL C00754 V=800.0 PL=0
MOVL C00755 V=800.0 PL=0
MOVL C00756 V=800.0 PL=0
MOVL C00757 V=800.0 PL=0
MOVL C00758 V=800.0 PL=0
MOVL C00759 V=800.0 PL=0
MOVL C00760 V=800.0 PL=0
MOVL C00761 V=800.0 PL=0
MOVL C00762 V=800.0 PL=0
MOVL C00763 V=800.0 PL=0
MOVL C00764 V=800.0 PL=0
MOVL C00765 V=800.0 PL=0
MOVL C00766 V=800.0 PL=0
MOVL C00767 V=800.0 PL=0
MOVL C00768 V=800.0 PL=0
MOVL C00769 V=800.0 PL=0
MOVL C00770 V=800.0 PL=0
MOVL C00771 V=800.0 PL=0
MOVL C00772 V=800.0 PL=0
MOVL C00773 V=800.0 PL=0
MOVL C00774 V=800.0 PL=0
MOVL C00775 V=800.0 PL=0
MOVL C00776 V=800.0 PL=0
MOVL C00777 V=800.0 PL=0
MOVL C00778 V=800.0 PL=0
MOVL C00779 V=800.0 PL=0
MOVL C00780 V=800.0 PL=0
MOVL C00781 V=800.0 PL=0
MOVL C00782 V=800.0 PL=0
MOVL C00783 V=800.0 PL=0
MOVL C00784 V=800.0 PL=0
MOVL C00785 V=800.0 PL=0
MOVL C00786 V=800.0 PL=0
MOVL C00787 V=800.0 PL=0
MOVL C00788 V=800.0 PL=0
MOVL C00789 V=800.0 PL=0
MOVL C00790 V=800.0 PL=0
MOVL C00791 V=800.0 PL=0
MOVL C00792 V=800.0 PL=0
MOVL C00793 V=800.0 PL=0
MOVL C00794 V=800.0 PL=0
MOVL C00795 V=800.0 PL=0
MOVL C00796 V=800.0 PL=0
MOVL C00797 V=800.0 PL=0
MOVL C00798 V=800.0 PL=0
MOVL C00799 V=800.0 PL=0
MOVL C00800 V=800.0 PL=0
MOVL C00801 V=800.0 PL=0
MOVL C00802 V=800.0 PL=0
MOVL C00803 V=800.0 PL=0
MOVL C00804 V=800.0 PL=0
MOVL C00805 V=800.0 PL=0
MOVL C00806 V=800.0 PL=0
MOVL C00807 V=800.0 PL=0
MOVL C00808 V=800.0 PL=0
MOVL C00809 V=800.0 PL=0
MOVL C00810 V=800.0 PL=0
MOVL C00811 V=800.0 PL=0
MOVL C00812 V=800.0 PL=0
MOVL C00813 V=800.0 PL=0
MOVL C00814 V=800.0 PL=0
MOVL C00815 V=800.0 PL=0
MOVL C00816 V=800.0 PL=0
MOVL C00817 V=800.0 PL=0
MOVL C00818 V=800.0 PL=0
MOVL C00819 V=800.0 PL=0
MOVL C00820 V=800.0 PL=0
MOVL C00821 V=800.0 PL=0
MOVL C00822 V=800.0 PL=0
MOVL C00823 V=800.0 PL=0
MOVL C00824 V=800.0 PL=0
MOVL C00825 V=800.0 PL=0
MOVL C00826 V=800.0 PL=0
MOVL C00827 V=800.0 PL=0
MOVL C00828 V=800.0 PL=0
MOVL C00829 V=800.0 PL=0
MOVL C00830 V=800.0 PL=0
MOVL C00831 V=800.0 PL=0
MOVL C00832 V=800.0 PL=0
MOVL C00833 V=800.0 PL=0
MOVL C00834 V=800.0 PL=0
MOVL C00835 V=800.0 PL=0
MOVL C00836 V=800.0 PL=0
MOVL C00837 V=800.0 PL=0
MOVL C00838 V=800.0 PL=0
MOVL C00839 V=800.0 PL=0
MOVL C00840 V=800.0 PL=0
MOVL C00841 V=800.0 PL=0
MOVL C00842 V=800.0 PL=0
MOVL C00843 V=800.0 PL=0
MOVL C00844 V=800.0 PL=0
MOVL C00845 V=800.0 PL=0
MOVL C00846 V=800.0 PL=0
MOVL C00847 V=800.0 PL=0
MOVL C00848 V=800.0 PL=0
MOVL C00849 V=800.0 PL=0
MOVL C00850 V=800.0 PL=0
MOVL C00851 V=800.0 PL=0
MOVL C00852 V=800.0 PL=0
MOVL C00853 V=800.0 PL=0
MOVL C00854 V=800.0 PL=0
MOVL C00855 V=800.0 PL=0
MOVL C00856 V=800.0 PL=0
MOVL C00857 V=800.0 PL=0
MOVL C00858 V=800.0 PL=0
MOVL C00859 V=800.0 PL=0
MOVL C00860 V=800.0 PL=0
MOVL C00861 V=800.0 PL=0
MOVL C00862 V=800.0 PL=0
MOVL C00863 V=800.0 PL=0
MOVL C00864 V=800.0 PL=0
MOVL C00865 V=800.0 PL=0
MOVL C00866 V=800.0 PL=0
MOVL C00867 V=800.0 PL=0
MOVL C00868 V=800.0 PL=0
MOVL C00869 V=800.0 PL=0
MOVL C00870 V=800.0 PL=0
MOVL C00871 V=800.0 PL=0
MOVL C00872 V=800.0 PL=0
MOVL C00873 V=800.0 PL=0
MOVL C00874 V=800.0 PL=0
MOVL C00875 V=800.0 PL=0
MOVL C00876 V=800.0 PL=0
MOVL C00877 V=800.0 PL=0
MOVL C00878 V=800.0 PL=0
MOVL C00879 V=800.0 PL=0
MOVL C00880 V=800.0 PL=0
MOVL C00881 V=800.0 PL=0
MOVL C00882 V=800.0 PL=0
MOVL C00883 V=800.0 PL=0
MOVL C00884 V=800.0 PL=0
MOVL C00885 V=800.0 PL=0
MOVL C00886 V=800.0 PL=0
MOVL C00887 V=800.0 PL=0
MOVL C00888 V=800.0 PL=0
MOVL C00889 V=800.0 PL=0
MOVL C00890 V=800.0 PL=0
MOVL C00891 V=800.0 PL=0
MOVL C00892 V=800.0 PL=0
MOVL C00893 V=800.0 PL=0
MOVL C00894 V=800.0 PL=0
MOVL C00895 V=800.0 PL=0
MOVL C00896 V=800.0 PL=0
MOVL C00897 V=800.0 PL=0
MOVL C00898 V=800.0 PL=0
MOVL C00899 V=800.0 PL=0
MOVL C00900 V=800.0 PL=0
MOVL C00901 V=800.0 PL=0
MOVL C00902 V=800.0 PL=0
MOVL C00903 V=800.0 PL=0
MOVL C00904 V=800.0 PL=0
MOVL C00905 V=800.0 PL=0
MOVL C00906 V=800.0 PL=0
MOVL C00907 V=800.0 PL=0
MOVL C00908 V=800.0 PL=0
MOVL C00909 V=800.0 PL=0
MOVL C00910 V=800.0 PL=0
MOVL C00911 V=800.0 PL=0
MOVL C00912 V=800.0 PL=0
MOVL C00913 V=800.0 PL=0
MOVL C00914 V=800.0 PL=0
MOVL C00915 V=800.0 PL=0
MOVL C00916 V=800.0 PL=0
MOVL C00917 V=800.0 PL=0
MOVL C00918 V=800.0 PL=0
MOVL C00919 V=800.0 PL=0
MOVL C00920 V=800.0 PL=0
MOVL C00921 V=800.0 PL=0
MOVL C00922 V=800.0 PL=0
MOVL C00923 V=800.0 PL=0
MOVL C00924 V=800.0 PL=0
MOVL C00925 V=800.0 PL=0
MOVL C00926 V=800.0 PL=0
MOVL C00927 V=800.0 PL=0
MOVL C00928 V=800.0 PL=0
MOVL C00929 V=800.0 PL=0
MOVL C00930 V=800.0 PL=0
MOVL C00931 V=800.0 PL=0
MOVL C00932 V=800.0 PL=0
MOVL C00933 V=800.0 PL=0
MOVL C00934 V=800.0 PL=0
MOVL C00935 V=800.0 PL=0
MOVL C00936 V=800.0 PL=0
MOVL C00937 V=800.0 PL=0
MOVL C00938 V=800.0 PL=0
MOVL C00939 V=800.0 PL=0
MOVL C00940 V=800.0 PL=0
MOVL C00941 V=800.0 PL=0
MOVL C00942 V=800.0 PL=0
MOVL C00943 V=800.0 PL=0
MOVL C00944 V=800.0 PL=0
MOVL C00945 V=800.0 PL=0
MOVL C00946 V=800.0 PL=0
MOVL C00947 V=800.0 PL=0
MOVL C00948 V=800.0 PL=0
MOVL C00949 V=800.0 PL=0
MOVL C00950 V=800.0 PL=0
MOVL C00951 V=800.0 PL=0
MOVL C00952 V=800.0 PL=0
MOVL C00953 V=800.0 PL=0
MOVL C00954 V=800.0 PL=0
MOVL C00955 V=800.0 PL=0
MOVL C00956 V=800.0 PL=0
MOVL C00957 V=800.0 PL=0
MOVL C00958 V=800.0 PL=0
MOVL C00959 V=800.0 PL=0
MOVL C00960 V=800.0 PL=0
MOVL C00961 V=800.0 PL=0
MOVL C00962 V=800.0 PL=0
MOVL C00963 V=800.0 PL=0
MOVL C00964 V=800.0 PL=0
MOVL C00965 V=800.0 PL=0
MOVL C00966 V=800.0 PL=0
MOVL C00967 V=800.0 PL=0
MOVL C00968 V=800.0 PL=0
MOVL C00969 V=800.0 PL=0
MOVL C00970 V=800.0 PL=0
MOVL C00971 V=800.0 PL=0
MOVL C00972 V=800.0 PL=0
MOVL C00973 V=800.0 PL=0
MOVL C00974 V=800.0 PL=0
MOVL C00975 V=800.0 PL=0
MOVL C00976 V=800.0 PL=0
MOVL C00977 V=800.0 PL=0
MOVL C00978 V=800.0 PL=0
MOVL C00979 V=800.0 PL=0
MOVL C00980 V=800.0 PL=0
MOVL C00981 V=800.0 PL=0
MOVL C00982 V=800.0 PL=0
MOVL C00983 V=800.0 PL=0
MOVL C00984 V=800.0 PL=0
MOVL C00985 V=800.0 PL=0
MOVL C00986 V=800.0 PL=0
MOVL C00987 V=800.0 PL=0
MOVL C00988 V=800.0 PL=0
MOVL C00989 V=800.0 PL=0
MOVL C00990 V=800.0 PL=0
MOVL C00991 V=800.0 PL=0
MOVL C00992 V=800.0 PL=0
MOVL C00993 V=800.0 PL=0
MOVL C00994 V=800.0 PL=0
MOVL C00995 V=800.0 PL=0
MOVL C00996 V=800.0 PL=0
MOVL C00997 V=800.0 PL=0
MOVL C00998 V=800.0 PL=0
MOVL C00999 V=800.0 PL=0
MOVL C01000 V=800.0 PL=0
MOVL C01001 V=800.0 PL=0
MOVL C01002 V=800.0 PL=0
MOVL C01003 V=800.0 PL=0
MOVL C01004 V=800.0 PL=0
MOVL C01005 V=800.0 PL=0
MOVL C01006 V=800.0 PL=0
MOVL C01007 V=800.0 PL=0
MOVL C01008 V=800.0 PL=0
MOVL C01009 V=800.0 PL=0
MOVL C01010 V=800.0 PL=0
MOVL C01011 V=800.0 PL=0
MOVL C01012 V=800.0 PL=0
MOVL C01013 V=800.0 PL=0
MOVL C01014 V=800.0 PL=0
MOVL C01015 V=800.0 PL=0
MOVL C01016 V=800.0 PL=0
MOVL C01017 V=800.0 PL=0
MOVL C01018 V=800.0 PL=0
MOVL C01019 V=800.0 PL=0
MOVL C01020 V=800.0 PL=0
MOVL C01021 V=800.0 PL=0
MOVL C01022 V=800.0 PL=0
MOVL C01023 V=800.0 PL=0
MOVL C01024 V=800.0 PL=0
MOVL C01025 V=800.0 PL=0
MOVL C01026 V=800.0 PL=0
MOVL C01027 V=800.0 PL=0
MOVL C01028 V=800.0 PL=0
MOVL C01029 V=800.0 PL=0
MOVL C01030 V=800.0 PL=0
MOVL C01031 V=800.0 PL=0
MOVL C01032 V=800.0 PL=0
MOVL C01033 V=800.0 PL=0
MOVL C01034 V=800.0 PL=0
MOVL C01035 V=800.0 PL=0
MOVL C01036 V=800.0 PL=0
MOVL C01037 V=800.0 PL=0
MOVL C01038 V=800.0 PL=0
MOVL C01039 V=800.0 PL=0
MOVL C01040 V=800.0 PL=0
MOVL C01041 V=800.0 PL=0
MOVL C01042 V=800.0 PL=0
MOVL C01043 V=800.0 PL=0
MOVL C01044 V=800.0 PL=0
MOVL C01045 V=800.0 PL=0
MOVL C01046 V=800.0 PL=0
MOVL C01047 V=800.0 PL=0
MOVL C01048 V=800.0 PL=0
MOVL C01049 V=800.0 PL=0
MOVL C01050 V=800.0 PL=0
MOVL C01051 V=800.0 PL=0
MOVL C01052 V=800.0 PL=0
MOVL C01053 V=800.0 PL=0
MOVL C01054 V=800.0 PL=0
MOVL C01055 V=800.0 PL=0
MOVL C01056 V=800.0 PL=0
MOVL C01057 V=800.0 PL=0
MOVL C01058 V=800.0 PL=0
MOVL C01059 V=800.0 PL=0
MOVL C01060 V=800.0 PL=0
MOVL C01061 V=800.0 PL=0
MOVL C01062 V=800.0 PL=0
MOVL C01063 V=800.0 PL=0
MOVL C01064 V=800.0 PL=0
MOVL C01065 V=800.0 PL=0
MOVL C01066 V=800.0 PL=0
MOVL C01067 V=800.0 PL=0
MOVL C01068 V=800.0 PL=0
MOVL C01069 V=800.0 PL=0
MOVL C01070 V=800.0 PL=0
MOVL C01071 V=800.0 PL=0
MOVL C01072 V=800.0 PL=0
MOVL C01073 V=800.0 PL=0
MOVL C01074 V=800.0 PL=0
MOVL C01075 V=800.0 PL=0
MOVL C01076 V=800.0 PL=0
MOVL C01077 V=800.0 PL=0
MOVL C01078 V=800.0 PL=0
MOVL C01079 V=800.0 PL=0
MOVL C01080 V=800.0 PL=0
MOVL C01081 V=800.0 PL=0
MOVL C01082 V=800.0 PL=0
MOVL C01083 V=800.0 PL=0
MOVL C01084 V=800.0 PL=0
MOVL C01085 V=800.0 PL=0
MOVL C01086 V=800.0 PL=0
MOVL C01087 V=800.0 PL=0
MOVL C01088 V=800.0 PL=0
MOVL C01089 V=800.0 PL=0
MOVL C01090 V=800.0 PL=0
MOVL C01091 V=800.0 PL=0
MOVL C01092 V=800.0 PL=0
MOVL C01093 V=800.0 PL=0
MOVL C01094 V=800.0 PL=0
MOVL C01095 V=800.0 PL=0
MOVL C01096 V=800.0 PL=0
MOVL C01097 V=800.0 PL=0
MOVL C01098 V=800.0 PL=0
MOVL C01099 V=800.0 PL=0
MOVL C01100 V=800.0 PL=0
MOVL C01101 V=800.0 PL=0
MOVL C01102 V=800.0 PL=0
MOVL C01103 V=800.0 PL=0
MOVL C01104 V=800.0 PL=0
MOVL C01105 V=800.0 PL=0
MOVL C01106 V=800.0 PL=0
MOVL C01107 V=800.0 PL=0
MOVL C01108 V=800.0 PL=0
MOVL C01109 V=800.0 PL=0
MOVL C01110 V=800.0 PL=0
MOVL C01111 V=800.0 PL=0
MOVL C01112 V=800.0 PL=0
MOVL C01113 V=800.0 PL=0
MOVL C01114 V=800.0 PL=0
MOVL C01115 V=800.0 PL=0
MOVL C01116 V=800.0 PL=0
MOVL C01117 V=800.0 PL=0
MOVL C01118 V=800.0 PL=0
MOVL C01119 V=800.0 PL=0
MOVL C01120 V=800.0 PL=0
MOVL C01121 V=800.0 PL=0
MOVL C01122 V=800.0 PL=0
MOVL C01123 V=800.0 PL=0
MOVL C01124 V=800.0 PL=0
MOVL C01125 V=800.0 PL=0
MOVL C01126 V=800.0 PL=0
MOVL C01127 V=800.0 PL=0
MOVL C01128 V=800.0 PL=0
MOVL C01129 V=800.0 PL=0
MOVL C01130 V=800.0 PL=0
MOVL C01131 V=800.0 PL=0
MOVL C01132 V=800.0 PL=0
MOVL C01133 V=800.0 PL=0
MOVL C01134 V=800.0 PL=0
MOVL C01135 V=800.0 PL=0
MOVL C01136 V=800.0 PL=0
MOVL C01137 V=800.0 PL=0
MOVL C01138 V=800.0 PL=0
MOVL C01139 V=800.0 PL=0
MOVL C01140 V=800.0 PL=0
MOVL C01141 V=800.0 PL=0
MOVL C01142 V=800.0 PL=0
MOVL C01143 V=800.0 PL=0
MOVL C01144 V=800.0 PL=0
MOVL C01145 V=800.0 PL=0
MOVL C01146 V=800.0 PL=0
MOVL C01147 V=800.0 PL=0
MOVL C01148 V=800.0 PL=0
MOVL C01149 V=800.0 PL=0
MOVL C01150 V=800.0 PL=0
MOVL C01151 V=800.0 PL=0
MOVL C01152 V=800.0 PL=0
MOVL C01153 V=800.0 PL=0
MOVL C01154 V=800.0 PL=0
MOVL C01155 V=800.0 PL=0
MOVL C01156 V=800.0 PL=0
MOVL C01157 V=800.0 PL=0
MOVL C01158 V=800.0 PL=0
MOVL C01159 V=800.0 PL=0
MOVL C01160 V=800.0 PL=0
MOVL C01161 V=800.0 PL=0
MOVL C01162 V=800.0 PL=0
MOVL C01163 V=800.0 PL=0
MOVL C01164 V=800.0 PL=0
MOVL C01165 V=800.0 PL=0
MOVL C01166 V=800.0 PL=0
MOVL C01167 V=800.0 PL=0
MOVL C01168 V=800.0 PL=0
MOVL C01169 V=800.0 PL=0
MOVL C01170 V=800.0 PL=0
MOVL C01171 V=800.0 PL=0
MOVL C01172 V=800.0 PL=0
MOVL C01173 V=800.0 PL=0
MOVL C01174 V=800.0 PL=0
MOVL C01175 V=800.0 PL=0
MOVL C01176 V=800.0 PL=0
MOVL C01177 V=800.0 PL=0
MOVL C01178 V=800.0 PL=0
MOVL C01179 V=800.0 PL=0
MOVL C01180 V=800.0 PL=0
MOVL C01181 V=800.0 PL=0
MOVL C01182 V=800.0 PL=0
MOVL C01183 V=800.0 PL=0
MOVL C01184 V=800.0 PL=0
MOVL C01185 V=800.0 PL=0
MOVL C01186 V=800.0 PL=0
MOVL C01187 V=800.0 PL=0
MOVL C01188 V=800.0 PL=0
MOVL C01189 V=800.0 PL=0
MOVL C01190 V=800.0 PL=0
MOVL C01191 V=800.0 PL=0
MOVL C01192 V=800.0 PL=0
MOVL C01193 V=800.0 PL=0
MOVL C01194 V=800.0 PL=0
MOVL C01195 V=800.0 PL=0
MOVL C01196 V=800.0 PL=0
MOVL C01197 V=800.0 PL=0
MOVL C01198 V=800.0 PL=0
MOVL C01199 V=800.0 PL=0
MOVL C01200 V=800.0 PL=0
MOVL C01201 V=800.0 PL=0
MOVL C01202 V=800.0 PL=0
MOVL C01203 V=800.0 PL=0
MOVL C01204 V=800.0 PL=0
MOVL C01205 V=800.0 PL=0
MOVL C01206 V=800.0 PL=0
MOVL C01207 V=800.0 PL=0
MOVL C01208 V=800.0 PL=0
MOVL C01209 V=800.0 PL=0
MOVL C01210 V=800.0 PL=0
MOVL C01211 V=800.0 PL=0
MOVL C01212 V=800.0 PL=0
MOVL C01213 V=800.0 PL=0
MOVL C01214 V=800.0 PL=0
MOVL C01215 V=800.0 PL=0
MOVL C01216 V=800.0 PL=0
MOVL C01217 V=800.0 PL=0
MOVL C01218 V=800.0 PL=0
MOVL C01219 V=800.0 PL=0
MOVL C01220 V=800.0 PL=0
MOVL C01221 V=800.0 PL=0
MOVL C01222 V=800.0 PL=0
MOVL C01223 V=800.0 PL=0
MOVL C01224 V=800.0 PL=0
MOVL C01225 V=800.0 PL=0
MOVL C01226 V=800.0 PL=0
MOVL C01227 V=800.0 PL=0
MOVL C01228 V=800.0 PL=0
MOVL C01229 V=800.0 PL=0
MOVL C01230 V=800.0 PL=0
MOVL C01231 V=800.0 PL=0
MOVL C01232 V=800.0 PL=0
MOVL C01233 V=800.0 PL=0
MOVL C01234 V=800.0 PL=0
MOVL C01235 V=800.0 PL=0
MOVL C01236 V=800.0 PL=0
MOVL C01237 V=800.0 PL=0
MOVL C01238 V=800.0 PL=0
MOVL C01239 V=800.0 PL=0
MOVL C01240 V=800.0 PL=0
MOVL C01241 V=800.0 PL=0
MOVL C01242 V=800.0 PL=0
MOVL C01243 V=800.0 PL=0
MOVL C01244 V=800.0 PL=0
MOVL C01245 V=800.0 PL=0
MOVL C01246 V=800.0 PL=0
MOVL C01247 V=800.0 PL=0
MOVL C01248 V=800.0 PL=0
MOVL C01249 V=800.0 PL=0
MOVL C01250 V=800.0 PL=0
MOVL C01251 V=800.0 PL=0
MOVL C01252 V=800.0 PL=0
MOVL C01253 V=800.0 PL=0
MOVL C01254 V=800.0 PL=0
MOVL C01255 V=800.0 PL=0
MOVL C01256 V=800.0 PL=0
MOVL C01257 V=800.0 PL=0
MOVL C01258 V=800.0 PL=0
MOVL C01259 V=800.0 PL=0
MOVL C01260 V=800.0 PL=0
MOVL C01261 V=800.0 PL=0
MOVL C01262 V=800.0 PL=0
MOVL C01263 V=800.0 PL=0
MOVL C01264 V=800.0 PL=0
MOVL C01265 V=800.0 PL=0
MOVL C01266 V=800.0 PL=0
MOVL C01267 V=800.0 PL=0
MOVL C01268 V=800.0 PL=0
MOVL C01269 V=800.0 PL=0
MOVL C01270 V=800.0 PL=0
MOVL C01271 V=800.0 PL=0
MOVL C01272 V=800.0 PL=0
MOVL C01273 V=800.0 PL=0
MOVL C01274 V=800.0 PL=0
MOVL C01275 V=800.0 PL=0
MOVL C01276 V=800.0 PL=0
MOVL C01277 V=800.0 PL=0
MOVL C01278 V=800.0 PL=0
MOVL C01279 V=800.0 PL=0
MOVL C01280 V=800.0 PL=0
MOVL C01281 V=800.0 PL=0
MOVL C01282 V=800.0 PL=0
MOVL C01283 V=800.0 PL=0
MOVL C01284 V=800.0 PL=0
MOVL C01285 V=800.0 PL=0
MOVL C01286 V=800.0 PL=0
MOVL C01287 V=800.0 PL=0
MOVL C01288 V=800.0 PL=0
MOVL C01289 V=800.0 PL=0
MOVL C01290 V=800.0 PL=0
MOVL C01291 V=800.0 PL=0
MOVL C01292 V=800.0 PL=0
MOVL C01293 V=800.0 PL=0
MOVL C01294 V=800.0 PL=0
MOVL C01295 V=800.0 PL=0
MOVL C01296 V=800.0 PL=0
MOVL C01297 V=800.0 PL=0
MOVL C01298 V=800.0 PL=0
MOVL C01299 V=800.0 PL=0
MOVL C01300 V=800.0 PL=0
MOVL C01301 V=800.0 PL=0
MOVL C01302 V=800.0 PL=0
MOVL C01303 V=800.0 PL=0
MOVL C01304 V=800.0 PL=0
MOVL C01305 V=800.0 PL=0
MOVL C01306 V=800.0 PL=0
MOVL C01307 V=800.0 PL=0
MOVL C01308 V=800.0 PL=0
MOVL C01309 V=800.0 PL=0
MOVL C01310 V=800.0 PL=0
MOVL C01311 V=800.0 PL=0
MOVL C01312 V=800.0 PL=0
MOVL C01313 V=800.0 PL=0
MOVL C01314 V=800.0 PL=0
MOVL C01315 V=800.0 PL=0
MOVL C01316 V=800.0 PL=0
MOVL C01317 V=800.0 PL=0
MOVL C01318 V=800.0 PL=0
MOVL C01319 V=800.0 PL=0
MOVL C01320 V=800.0 PL=0
MOVL C01321 V=800.0 PL=0
MOVL C01322 V=800.0 PL=0
MOVL C01323 V=800.0 PL=0
MOVL C01324 V=800.0 PL=0
MOVL C01325 V=800.0 PL=0
MOVL C01326 V=800.0 PL=0
MOVL C01327 V=800.0 PL=0
MOVL C01328 V=800.0 PL=0
MOVL C01329 V=800.0 PL=0
MOVL C01330 V=800.0 PL=0
MOVL C01331 V=800.0 PL=0
MOVL C01332 V=800.0 PL=0
MOVL C01333 V=800.0 PL=0
MOVL C01334 V=800.0 PL=0
MOVL C01335 V=800.0 PL=0
MOVL C01336 V=800.0 PL=0
MOVL C01337 V=800.0 PL=0
MOVL C01338 V=800.0 PL=0
MOVL C01339 V=800.0 PL=0
MOVL C01340 V=800.0 PL=0
MOVL C01341 V=800.0 PL=0
MOVL C01342 V=800.0 PL=0
MOVL C01343 V=800.0 PL=0
MOVL C01344 V=800.0 PL=0
MOVL C01345 V=800.0 PL=0
MOVL C01346 V=800.0 PL=0
MOVL C01347 V=800.0 PL=0
MOVL C01348 V=800.0 PL=0
MOVL C01349 V=800.0 PL=0
MOVL C01350 V=800.0 PL=0
MOVL C01351 V=800.0 PL=0
MOVL C01352 V=800.0 PL=0
MOVL C01353 V=800.0 PL=0
MOVL C01354 V=800.0 PL=0
MOVL C01355 V=800.0 PL=0
MOVL C01356 V=800.0 PL=0
MOVL C01357 V=800.0 PL=0
MOVL C01358 V=800.0 PL=0
MOVL C01359 V=800.0 PL=0
MOVL C01360 V=800.0 PL=0
MOVL C01361 V=800.0 PL=0
MOVL C01362 V=800.0 PL=0
MOVL C01363 V=800.0 PL=0
MOVL C01364 V=800.0 PL=0
MOVL C01365 V=800.0 PL=0
MOVL C01366 V=800.0 PL=0
MOVL C01367 V=800.0 PL=0
MOVL C01368 V=800.0 PL=0
MOVL C01369 V=800.0 PL=0
MOVL C01370 V=800.0 PL=0
MOVL C01371 V=800.0 PL=0
MOVL C01372 V=800.0 PL=0
MOVL C01373 V=800.0 PL=0
MOVL C01374 V=800.0 PL=0
MOVL C01375 V=800.0 PL=0
MOVL C01376 V=800.0 PL=0
MOVL C01377 V=800.0 PL=0
MOVL C01378 V=800.0 PL=0
MOVL C01379 V=800.0 PL=0
MOVL C01380 V=800.0 PL=0
MOVL C01381 V=800.0 PL=0
MOVL C01382 V=800.0 PL=0
MOVL C01383 V=800.0 PL=0
MOVL C01384 V=800.0 PL=0
MOVL C01385 V=800.0 PL=0
MOVL C01386 V=800.0 PL=0
MOVL C01387 V=800.0 PL=0
MOVL C01388 V=800.0 PL=0
MOVL C01389 V=800.0 PL=0
MOVL C01390 V=800.0 PL=0
MOVL C01391 V=800.0 PL=0
MOVL C01392 V=800.0 PL=0
MOVL C01393 V=800.0 PL=0
MOVL C01394 V=800.0 PL=0
MOVL C01395 V=800.0 PL=0
MOVL C01396 V=800.0 PL=0
MOVL C01397 V=800.0 PL=0
MOVL C01398 V=800.0 PL=0
MOVL C01399 V=800.0 PL=0
MOVL C01400 V=800.0 PL=0
MOVL C01401 V=800.0 PL=0
MOVL C01402 V=800.0 PL=0
MOVL C01403 V=800.0 PL=0
MOVL C01404 V=800.0 PL=0
MOVL C01405 V=800.0 PL=0
MOVL C01406 V=800.0 PL=0
MOVL C01407 V=800.0 PL=0
MOVL C01408 V=800.0 PL=0
MOVL C01409 V=800.0 PL=0
MOVL C01410 V=800.0 PL=0
MOVL C01411 V=800.0 PL=0
MOVL C01412 V=800.0 PL=0
MOVL C01413 V=800.0 PL=0
MOVL C01414 V=800.0 PL=0
MOVL C01415 V=800.0 PL=0
MOVL C01416 V=800.0 PL=0
MOVL C01417 V=800.0 PL=0
MOVL C01418 V=800.0 PL=0
MOVL C01419 V=800.0 PL=0
MOVL C01420 V=800.0 PL=0
MOVL C01421 V=800.0 PL=0
MOVL C01422 V=800.0 PL=0
MOVL C01423 V=800.0 PL=0
MOVL C01424 V=800.0 PL=0
MOVL C01425 V=800.0 PL=0
MOVL C01426 V=800.0 PL=0
MOVL C01427 V=800.0 PL=0
MOVL C01428 V=800.0 PL=0
MOVL C01429 V=800.0 PL=0
MOVL C01430 V=800.0 PL=0
MOVL C01431 V=800.0 PL=0
MOVL C01432 V=800.0 PL=0
MOVL C01433 V=800.0 PL=0
MOVL C01434 V=800.0 PL=0
MOVL C01435 V=800.0 PL=0
MOVL C01436 V=800.0 PL=0
MOVL C01437 V=800.0 PL=0
MOVL C01438 V=800.0 PL=0
MOVL C01439 V=800.0 PL=0
MOVL C01440 V=800.0 PL=0
MOVL C01441 V=800.0 PL=0
MOVL C01442 V=800.0 PL=0
MOVL C01443 V=800.0 PL=0
MOVL C01444 V=800.0 PL=0
MOVL C01445 V=800.0 PL=0
MOVL C01446 V=800.0 PL=0
MOVL C01447 V=800.0 PL=0
MOVL C01448 V=800.0 PL=0
MOVL C01449 V=800.0 PL=0
MOVL C01450 V=800.0 PL=0
MOVL C01451 V=800.0 PL=0
MOVL C01452 V=800.0 PL=0
MOVL C01453 V=800.0 PL=0
MOVL C01454 V=800.0 PL=0
MOVL C01455 V=800.0 PL=0
MOVL C01456 V=800.0 PL=0
MOVL C01457 V=800.0 PL=0
MOVL C01458 V=800.0 PL=0
MOVL C01459 V=800.0 PL=0
MOVL C01460 V=800.0 PL=0
MOVL C01461 V=800.0 PL=0
MOVL C01462 V=800.0 PL=0
MOVL C01463 V=800.0 PL=0
MOVL C01464 V=800.0 PL=0
MOVL C01465 V=800.0 PL=0
MOVL C01466 V=800.0 PL=0
MOVL C01467 V=800.0 PL=0
MOVL C01468 V=800.0 PL=0
MOVL C01469 V=800.0 PL=0
MOVL C01470 V=800.0 PL=0
MOVL C01471 V=800.0 PL=0
MOVL C01472 V=800.0 PL=0
MOVL C01473 V=800.0 PL=0
MOVL C01474 V=800.0 PL=0
MOVL C01475 V=800.0 PL=0
MOVL C01476 V=800.0 PL=0
MOVL C01477 V=800.0 PL=0
MOVL C01478 V=800.0 PL=0
MOVL C01479 V=800.0 PL=0
MOVL C01480 V=800.0 PL=0
MOVL C01481 V=800.0 PL=0
MOVL C01482 V=800.0 PL=0
MOVL C01483 V=800.0 PL=0
MOVL C01484 V=800.0 PL=0
MOVL C01485 V=800.0 PL=0
MOVL C01486 V=800.0 PL=0
MOVL C01487 V=800.0 PL=0
MOVL C01488 V=800.0 PL=0
MOVL C01489 V=800.0 PL=0
MOVL C01490 V=800.0 PL=0
MOVL C01491 V=800.0 PL=0
MOVL C01492 V=800.0 PL=0
MOVL C01493 V=800.0 PL=0
MOVL C01494 V=800.0 PL=0
MOVL C01495 V=800.0 PL=0
MOVL C01496 V=800.0 PL=0
MOVL C01497 V=800.0 PL=0
MOVL C01498 V=800.0 PL=0
MOVL C01499 V=800.0 PL=0
MOVL C01500 V=800.0 PL=0
MOVL C01501 V=800.0 PL=0
MOVL C01502 V=800.0 PL=0
MOVL C01503 V=800.0 PL=0
MOVL C01504 V=800.0 PL=0
MOVL C01505 V=800.0 PL=0
MOVL C01506 V=800.0 PL=0
MOVL C01507 V=800.0 PL=0
MOVL C01508 V=800.0 PL=0
MOVL C01509 V=800.0 PL=0
MOVL C01510 V=800.0 PL=0
MOVL C01511 V=800.0 PL=0
MOVL C01512 V=800.0 PL=0
MOVL C01513 V=800.0 PL=0
MOVL C01514 V=800.0 PL=0
MOVL C01515 V=800.0 PL=0
MOVL C01516 V=800.0 PL=0
MOVL C01517 V=800.0 PL=0
MOVL C01518 V=800.0 PL=0
MOVL C01519 V=800.0 PL=0
MOVL C01520 V=800.0 PL=0
MOVL C01521 V=800.0 PL=0
MOVL C01522 V=800.0 PL=0
MOVL C01523 V=800.0 PL=0
MOVL C01524 V=800.0 PL=0
MOVL C01525 V=800.0 PL=0
MOVL C01526 V=800.0 PL=0
MOVL C01527 V=800.0 PL=0
MOVL C01528 V=800.0 PL=0
MOVL C01529 V=800.0 PL=0
MOVL C01530 V=800.0 PL=0
MOVL C01531 V=800.0 PL=0
MOVL C01532 V=800.0 PL=0
MOVL C01533 V=800.0 PL=0
MOVL C01534 V=800.0 PL=0
MOVL C01535 V=800.0 PL=0
MOVL C01536 V=800.0 PL=0
MOVL C01537 V=800.0 PL=0
MOVL C01538 V=800.0 PL=0
MOVL C01539 V=800.0 PL=0
MOVL C01540 V=800.0 PL=0
MOVL C01541 V=800.0 PL=0
MOVL C01542 V=800.0 PL=0
MOVL C01543 V=800.0 PL=0
MOVL C01544 V=800.0 PL=0
MOVL C01545 V=800.0 PL=0
MOVL C01546 V=800.0 PL=0
MOVL C01547 V=800.0 PL=0
MOVL C01548 V=800.0 PL=0
MOVL C01549 V=800.0 PL=0
MOVL C01550 V=800.0 PL=0
MOVL C01551 V=800.0 PL=0
MOVL C01552 V=800.0 PL=0
MOVL C01553 V=800.0 PL=0
MOVL C01554 V=800.0 PL=0
MOVL C01555 V=800.0 PL=0
MOVL C01556 V=800.0 PL=0
MOVL C01557 V=800.0 PL=0
MOVL C01558 V=800.0 PL=0
MOVL C01559 V=800.0 PL=0
MOVL C01560 V=800.0 PL=0
MOVL C01561 V=800.0 PL=0
MOVL C01562 V=800.0 PL=0
MOVL C01563 V=800.0 PL=0
MOVL C01564 V=800.0 PL=0
MOVL C01565 V=800.0 PL=0
MOVL C01566 V=800.0 PL=0
MOVL C01567 V=800.0 PL=0
MOVL C01568 V=800.0 PL=0
MOVL C01569 V=800.0 PL=0
MOVL C01570 V=800.0 PL=0
MOVL C01571 V=800.0 PL=0
MOVL C01572 V=800.0 PL=0
MOVL C01573 V=800.0 PL=0
MOVL C01574 V=800.0 PL=0
MOVL C01575 V=800.0 PL=0
MOVL C01576 V=800.0 PL=0
MOVL C01577 V=800.0 PL=0
MOVL C01578 V=800.0 PL=0
MOVL C01579 V=800.0 PL=0
MOVL C01580 V=800.0 PL=0
MOVL C01581 V=800.0 PL=0
MOVL C01582 V=800.0 PL=0
MOVL C01583 V=800.0 PL=0
MOVL C01584 V=800.0 PL=0
MOVL C01585 V=800.0 PL=0
MOVL C01586 V=800.0 PL=0
MOVL C01587 V=800.0 PL=0
MOVL C01588 V=800.0 PL=0
MOVL C01589 V=800.0 PL=0
MOVL C01590 V=800.0 PL=0
MOVL C01591 V=800.0 PL=0
MOVL C01592 V=800.0 PL=0
MOVL C01593 V=800.0 PL=0
MOVL C01594 V=800.0 PL=0
MOVL C01595 V=800.0 PL=0
MOVL C01596 V=800.0 PL=0
MOVL C01597 V=800.0 PL=0
MOVL C01598 V=800.0 PL=0
MOVL C01599 V=800.0 PL=0
MOVL C01600 V=800.0 PL=0
MOVL C01601 V=800.0 PL=0
MOVL C01602 V=800.0 PL=0
MOVL C01603 V=800.0 PL=0
MOVL C01604 V=800.0 PL=0
MOVL C01605 V=800.0 PL=0
MOVL C01606 V=800.0 PL=0
MOVL C01607 V=800.0 PL=0
MOVL C01608 V=800.0 PL=0
MOVL C01609 V=800.0 PL=0
MOVL C01610 V=800.0 PL=0
MOVL C01611 V=800.0 PL=0
MOVL C01612 V=800.0 PL=0
MOVL C01613 V=800.0 PL=0
MOVL C01614 V=800.0 PL=0
MOVL C01615 V=800.0 PL=0
MOVL C01616 V=800.0 PL=0
MOVL C01617 V=800.0 PL=0
MOVL C01618 V=800.0 PL=0
MOVL C01619 V=800.0 PL=0
MOVL C01620 V=800.0 PL=0
MOVL C01621 V=800.0 PL=0
MOVL C01622 V=800.0 PL=0
MOVL C01623 V=800.0 PL=0
MOVL C01624 V=800.0 PL=0
MOVL C01625 V=800.0 PL=0
MOVL C01626 V=800.0 PL=0
MOVL C01627 V=800.0 PL=0
MOVL C01628 V=800.0 PL=0
MOVL C01629 V=800.0 PL=0
MOVL C01630 V=800.0 PL=0
MOVL C01631 V=800.0 PL=0
MOVL C01632 V=800.0 PL=0
MOVL C01633 V=800.0 PL=0
MOVL C01634 V=800.0 PL=0
MOVL C01635 V=800.0 PL=0
MOVL C01636 V=800.0 PL=0
MOVL C01637 V=800.0 PL=0
MOVL C01638 V=800.0 PL=0
MOVL C01639 V=800.0 PL=0
MOVL C01640 V=800.0 PL=0
MOVL C01641 V=800.0 PL=0
MOVL C01642 V=800.0 PL=0
MOVL C01643 V=800.0 PL=0
MOVL C01644 V=800.0 PL=0
MOVL C01645 V=800.0 PL=0
MOVL C01646 V=800.0 PL=0
MOVL C01647 V=800.0 PL=0
MOVL C01648 V=800.0 PL=0
MOVL C01649 V=800.0 PL=0
MOVL C01650 V=800.0 PL=0
MOVL C01651 V=800.0 PL=0
MOVL C01652 V=800.0 PL=0
MOVL C01653 V=800.0 PL=0
MOVL C01654 V=800.0 PL=0
MOVL C01655 V=800.0 PL=0
MOVL C01656 V=800.0 PL=0
MOVL C01657 V=800.0 PL=0
MOVL C01658 V=800.0 PL=0
MOVL C01659 V=800.0 PL=0
MOVL C01660 V=800.0 PL=0
MOVL C01661 V=800.0 PL=0
MOVL C01662 V=800.0 PL=0
MOVL C01663 V=800.0 PL=0
MOVL C01664 V=800.0 PL=0
MOVL C01665 V=800.0 PL=0
MOVL C01666 V=800.0 PL=0
MOVL C01667 V=800.0 PL=0
MOVL C01668 V=800.0 PL=0
MOVL C01669 V=800.0 PL=0
MOVL C01670 V=800.0 PL=0
MOVL C01671 V=800.0 PL=0
MOVL C01672 V=800.0 PL=0
MOVL C01673 V=800.0 PL=0
MOVL C01674 V=800.0 PL=0
MOVL C01675 V=800.0 PL=0
MOVL C01676 V=800.0 PL=0
MOVL C01677 V=800.0 PL=0
MOVL C01678 V=800.0 PL=0
MOVL C01679 V=800.0 PL=0
MOVL C01680 V=800.0 PL=0
MOVL C01681 V=800.0 PL=0
MOVL C01682 V=800.0 PL=0
MOVL C01683 V=800.0 PL=0
MOVL C01684 V=800.0 PL=0
MOVL C01685 V=800.0 PL=0
MOVL C01686 V=800.0 PL=0
MOVL C01687 V=800.0 PL=0
MOVL C01688 V=800.0 PL=0
MOVL C01689 V=800.0 PL=0
MOVL C01690 V=800.0 PL=0
MOVL C01691 V=800.0 PL=0
MOVL C01692 V=800.0 PL=0
MOVL C01693 V=800.0 PL=0
MOVL C01694 V=800.0 PL=0
MOVL C01695 V=800.0 PL=0
MOVL C01696 V=800.0 PL=0
MOVL C01697 V=800.0 PL=0
MOVL C01698 V=800.0 PL=0
MOVL C01699 V=800.0 PL=0
MOVL C01700 V=800.0 PL=0
MOVL C01701 V=800.0 PL=0
MOVL C01702 V=800.0 PL=0
MOVL C01703 V=800.0 PL=0
MOVL C01704 V=800.0 PL=0
MOVL C01705 V=800.0 PL=0
MOVL C01706 V=800.0 PL=0
MOVL C01707 V=800.0 PL=0
MOVL C01708 V=800.0 PL=0
MOVL C01709 V=800.0 PL=0
MOVL C01710 V=800.0 PL=0
MOVL C01711 V=800.0 PL=0
MOVL C01712 V=800.0 PL=0
MOVL C01713 V=800.0 PL=0
MOVL C01714 V=800.0 PL=0
MOVL C01715 V=800.0 PL=0
MOVL C01716 V=800.0 PL=0
MOVL C01717 V=800.0 PL=0
MOVL C01718 V=800.0 PL=0
MOVL C01719 V=800.0 PL=0
MOVL C01720 V=800.0 PL=0
MOVL C01721 V=800.0 PL=0
MOVL C01722 V=800.0 PL=0
MOVL C01723 V=800.0 PL=0
MOVL C01724 V=800.0 PL=0
MOVL C01725 V=800.0 PL=0
MOVL C01726 V=800.0 PL=0
MOVL C01727 V=800.0 PL=0
MOVL C01728 V=800.0 PL=0
MOVL C01729 V=800.0 PL=0
MOVL C01730 V=800.0 PL=0
MOVL C01731 V=800.0 PL=0
MOVL C01732 V=800.0 PL=0
MOVL C01733 V=800.0 PL=0
MOVL C01734 V=800.0 PL=0
MOVL C01735 V=800.0 PL=0
MOVL C01736 V=800.0 PL=0
MOVL C01737 V=800.0 PL=0
MOVL C01738 V=800.0 PL=0
MOVL C01739 V=800.0 PL=0
MOVL C01740 V=800.0 PL=0
MOVL C01741 V=800.0 PL=0
MOVL C01742 V=800.0 PL=0
MOVL C01743 V=800.0 PL=0
MOVL C01744 V=800.0 PL=0
MOVL C01745 V=800.0 PL=0
MOVL C01746 V=800.0 PL=0
MOVL C01747 V=800.0 PL=0
MOVL C01748 V=800.0 PL=0
MOVL C01749 V=800.0 PL=0
MOVL C01750 V=800.0 PL=0
MOVL C01751 V=800.0 PL=0
MOVL C01752 V=800.0 PL=0
MOVL C01753 V=800.0 PL=0
MOVL C01754 V=800.0 PL=0
MOVL C01755 V=800.0 PL=0
MOVL C01756 V=800.0 PL=0
MOVL C01757 V=800.0 PL=0
MOVL C01758 V=800.0 PL=0
MOVL C01759 V=800.0 PL=0
MOVL C01760 V=800.0 PL=0
MOVL C01761 V=800.0 PL=0
MOVL C01762 V=800.0 PL=0
MOVL C01763 V=800.0 PL=0
MOVL C01764 V=800.0 PL=0
MOVL C01765 V=800.0 PL=0
MOVL C01766 V=800.0 PL=0
MOVL C01767 V=800.0 PL=0
MOVL C01768 V=800.0 PL=0
MOVL C01769 V=800.0 PL=0
MOVL C01770 V=800.0 PL=0
MOVL C01771 V=800.0 PL=0
MOVL C01772 V=800.0 PL=0
MOVL C01773 V=800.0 PL=0
MOVL C01774 V=800.0 PL=0
MOVL C01775 V=800.0 PL=0
MOVL C01776 V=800.0 PL=0
MOVL C01777 V=800.0 PL=0
MOVL C01778 V=800.0 PL=0
MOVL C01779 V=800.0 PL=0
MOVL C01780 V=800.0 PL=0
MOVL C01781 V=800.0 PL=0
MOVL C01782 V=800.0 PL=0
MOVL C01783 V=800.0 PL=0
MOVL C01784 V=800.0 PL=0
MOVL C01785 V=800.0 PL=0
MOVL C01786 V=800.0 PL=0
MOVL C01787 V=800.0 PL=0
MOVL C01788 V=800.0 PL=0
MOVL C01789 V=800.0 PL=0
MOVL C01790 V=800.0 PL=0
MOVL C01791 V=800.0 PL=0
MOVL C01792 V=800.0 PL=0
MOVL C01793 V=800.0 PL=0
MOVL C01794 V=800.0 PL=0
MOVL C01795 V=800.0 PL=0
MOVL C01796 V=800.0 PL=0
MOVL C01797 V=800.0 PL=0
MOVL C01798 V=800.0 PL=0
MOVL C01799 V=800.0 PL=0
MOVL C01800 V=800.0 PL=0
MOVL C01801 V=800.0 PL=0
MOVL C01802 V=800.0 PL=0
MOVL C01803 V=800.0 PL=0
MOVL C01804 V=800.0 PL=0
MOVL C01805 V=800.0 PL=0
MOVL C01806 V=800.0 PL=0
MOVL C01807 V=800.0 PL=0
MOVL C01808 V=800.0 PL=0
MOVL C01809 V=800.0 PL=0
MOVL C01810 V=800.0 PL=0
MOVL C01811 V=800.0 PL=0
MOVL C01812 V=800.0 PL=0
MOVL C01813 V=800.0 PL=0
MOVL C01814 V=800.0 PL=0
MOVL C01815 V=800.0 PL=0
MOVL C01816 V=800.0 PL=0
MOVL C01817 V=800.0 PL=0
MOVL C01818 V=800.0 PL=0
MOVL C01819 V=800.0 PL=0
MOVL C01820 V=800.0 PL=0
MOVL C01821 V=800.0 PL=0
MOVL C01822 V=800.0 PL=0
MOVL C01823 V=800.0 PL=0
MOVL C01824 V=800.0 PL=0
MOVL C01825 V=800.0 PL=0
MOVL C01826 V=800.0 PL=0
MOVL C01827 V=800.0 PL=0
MOVL C01828 V=800.0 PL=0
MOVL C01829 V=800.0 PL=0
MOVL C01830 V=800.0 PL=0
MOVL C01831 V=800.0 PL=0
MOVL C01832 V=800.0 PL=0
MOVL C01833 V=800.0 PL=0
MOVL C01834 V=800.0 PL=0
MOVL C01835 V=800.0 PL=0
MOVL C01836 V=800.0 PL=0
MOVL C01837 V=800.0 PL=0
MOVL C01838 V=800.0 PL=0
MOVL C01839 V=800.0 PL=0
MOVL C01840 V=800.0 PL=0
MOVL C01841 V=800.0 PL=0
MOVL C01842 V=800.0 PL=0
MOVL C01843 V=800.0 PL=0
MOVL C01844 V=800.0 PL=0
MOVL C01845 V=800.0 PL=0
MOVL C01846 V=800.0 PL=0
MOVL C01847 V=800.0 PL=0
MOVL C01848 V=800.0 PL=0
MOVL C01849 V=800.0 PL=0
MOVL C01850 V=800.0 PL=0
MOVL C01851 V=800.0 PL=0
MOVL C01852 V=800.0 PL=0
MOVL C01853 V=800.0 PL=0
MOVL C01854 V=800.0 PL=0
MOVL C01855 V=800.0 PL=0
MOVL C01856 V=800.0 PL=0
MOVL C01857 V=800.0 PL=0
MOVL C01858 V=800.0 PL=0
MOVL C01859 V=800.0 PL=0
MOVL C01860 V=800.0 PL=0
MOVL C01861 V=800.0 PL=0
MOVL C01862 V=800.0 PL=0
MOVL C01863 V=800.0 PL=0
MOVL C01864 V=800.0 PL=0
MOVL C01865 V=800.0 PL=0
MOVL C01866 V=800.0 PL=0
MOVL C01867 V=800.0 PL=0
MOVL C01868 V=800.0 PL=0
MOVL C01869 V=800.0 PL=0
MOVL C01870 V=800.0 PL=0
MOVL C01871 V=800.0 PL=0
MOVL C01872 V=800.0 PL=0
MOVL C01873 V=800.0 PL=0
MOVL C01874 V=800.0 PL=0
MOVL C01875 V=800.0 PL=0
MOVL C01876 V=800.0 PL=0
MOVL C01877 V=800.0 PL=0
MOVL C01878 V=800.0 PL=0
MOVL C01879 V=800.0 PL=0
MOVL C01880 V=800.0 PL=0
MOVL C01881 V=800.0 PL=0
MOVL C01882 V=800.0 PL=0
MOVL C01883 V=800.0 PL=0
MOVL C01884 V=800.0 PL=0
MOVL C01885 V=800.0 PL=0
MOVL C01886 V=800.0 PL=0
MOVL C01887 V=800.0 PL=0
MOVL C01888 V=800.0 PL=0
MOVL C01889 V=800.0 PL=0
MOVL C01890 V=800.0 PL=0
MOVL C01891 V=800.0 PL=0
MOVL C01892 V=800.0 PL=0
MOVL C01893 V=800.0 PL=0
MOVL C01894 V=800.0 PL=0
MOVL C01895 V=800.0 PL=0
MOVL C01896 V=800.0 PL=0
MOVL C01897 V=800.0 PL=0
MOVL C01898 V=800.0 PL=0
MOVL C01899 V=800.0 PL=0
MOVL C01900 V=800.0 PL=0
MOVL C01901 V=800.0 PL=0
MOVL C01902 V=800.0 PL=0
MOVL C01903 V=800.0 PL=0
MOVL C01904 V=800.0 PL=0
MOVL C01905 V=800.0 PL=0
MOVL C01906 V=800.0 PL=0
MOVL C01907 V=800.0 PL=0
MOVL C01908 V=800.0 PL=0
MOVL C01909 V=800.0 PL=0
MOVL C01910 V=800.0 PL=0
MOVL C01911 V=800.0 PL=0
MOVL C01912 V=800.0 PL=0
MOVL C01913 V=800.0 PL=0
MOVL C01914 V=800.0 PL=0
MOVL C01915 V=800.0 PL=0
MOVL C01916 V=800.0 PL=0
MOVL C01917 V=800.0 PL=0
MOVL C01918 V=800.0 PL=0
MOVL C01919 V=800.0 PL=0
MOVL C01920 V=800.0 PL=0
MOVL C01921 V=800.0 PL=0
MOVL C01922 V=800.0 PL=0
MOVL C01923 V=800.0 PL=0
MOVL C01924 V=800.0 PL=0
MOVL C01925 V=800.0 PL=0
MOVL C01926 V=800.0 PL=0
MOVL C01927 V=800.0 PL=0
MOVL C01928 V=800.0 PL=0
MOVL C01929 V=800.0 PL=0
MOVL C01930 V=800.0 PL=0
MOVL C01931 V=800.0 PL=0
MOVL C01932 V=800.0 PL=0
MOVL C01933 V=800.0 PL=0
MOVL C01934 V=800.0 PL=0
MOVL C01935 V=800.0 PL=0
MOVL C01936 V=800.0 PL=0
MOVL C01937 V=800.0 PL=0
MOVL C01938 V=800.0 PL=0
MOVL C01939 V=800.0 PL=0
MOVL C01940 V=800.0 PL=0
MOVL C01941 V=800.0 PL=0
MOVL C01942 V=800.0 PL=0
MOVL C01943 V=800.0 PL=0
MOVL C01944 V=800.0 PL=0
MOVL C01945 V=800.0 PL=0
MOVL C01946 V=800.0 PL=0
MOVL C01947 V=800.0 PL=0
MOVL C01948 V=800.0 PL=0
MOVL C01949 V=800.0 PL=0
MOVL C01950 V=800.0 PL=0
MOVL C01951 V=800.0 PL=0
MOVL C01952 V=800.0 PL=0
MOVL C01953 V=800.0 PL=0
MOVL C01954 V=800.0 PL=0
MOVL C01955 V=800.0 PL=0
MOVL C01956 V=800.0 PL=0
MOVL C01957 V=800.0 PL=0
MOVL C01958 V=800.0 PL=0
MOVL C01959 V=800.0 PL=0
MOVL C01960 V=800.0 PL=0
MOVL C01961 V=800.0 PL=0
MOVL C01962 V=800.0 PL=0
MOVL C01963 V=800.0 PL=0
MOVL C01964 V=800.0 PL=0
MOVL C01965 V=800.0 PL=0
MOVL C01966 V=800.0 PL=0
MOVL C01967 V=800.0 PL=0
MOVL C01968 V=800.0 PL=0
MOVL C01969 V=800.0 PL=0
MOVL C01970 V=800.0 PL=0
MOVL C01971 V=800.0 PL=0
MOVL C01972 V=800.0 PL=0
MOVL C01973 V=800.0 PL=0
MOVL C01974 V=800.0 PL=0
MOVL C01975 V=800.0 PL=0
MOVL C01976 V=800.0 PL=0
MOVL C01977 V=800.0 PL=0
MOVL C01978 V=800.0 PL=0
MOVL C01979 V=800.0 PL=0
MOVL C01980 V=800.0 PL=0
MOVL C01981 V=800.0 PL=0
MOVL C01982 V=800.0 PL=0
MOVL C01983 V=800.0 PL=0
MOVL C01984 V=800.0 PL=0
MOVL C01985 V=800.0 PL=0
MOVL C01986 V=800.0 PL=0
MOVL C01987 V=800.0 PL=0
MOVL C01988 V=800.0 PL=0
MOVL C01989 V=800.0 PL=0
MOVL C01990 V=800.0 PL=0
MOVL C01991 V=800.0 PL=0
MOVL C01992 V=800.0 PL=0
MOVL C01993 V=800.0 PL=0
MOVL C01994 V=800.0 PL=0
MOVL C01995 V=800.0 PL=0
MOVL C01996 V=800.0 PL=0
MOVL C01997 V=800.0 PL=0
MOVL C01998 V=800.0 PL=0
MOVL C01999 V=800.0 PL=0
MOVL C02000 V=800.0 PL=0
MOVL C02001 V=800.0 PL=0
MOVL C02002 V=800.0 PL=0
MOVL C02003 V=800.0 PL=0
MOVL C02004 V=800.0 PL=0
MOVL C02005 V=800.0 PL=0
MOVL C02006 V=800.0 PL=0
